               IF "MAX_VFDS" <> "MAX_ROOMS" * "MAX_RACKS_PER_ROOM" THEN
                   #bSettingsValid := FALSE;
                   #Status.ErrorMsg := CONCAT(IN1 := #Status.ErrorMsg, IN2 := ' MAX_VFDS != MAX_ROOMS*MAX_RACKS ');
               END_IF;

               IF #Controls.iSetNumRooms > "MAX_ROOMS" THEN
                   #bSettingsValid := FALSE;
                   #Status.ErrorMsg := CONCAT(IN1 := #Status.ErrorMsg, IN2 := ' NumRooms > MAX ');
               END_IF;

               FOR #i := 1 TO UINT_TO_INT("MAX_ROOMS") DO
                   IF #Controls.arrSetNumRacksPerRoom[#i] > "MAX_RACKS_PER_ROOM" THEN
                       #bSettingsValid := FALSE;
                       #Status.ErrorMsg := CONCAT(IN1 := #Status.ErrorMsg, IN2 := ' NumRacks > MAX ');
                       EXIT;
                   END_IF;
               END_FOR;

               IF "MAX_AI_PER_ROOM" <> ("NUM_AI_ROOM" + "NUM_AI_RACK" * "MAX_RACKS_PER_ROOM" + "EXTRA_AI_PER_ROOM") OR ( "MAX_AI_PER_ROOM" MOD 4 <> 0) THEN
                   #bSettingsValid := FALSE;
                   #Status.ErrorMsg := CONCAT(IN1 := #Status.ErrorMsg, IN2 := ' MAX_AI_PER_ROOM incorrect ');
               END_IF;

               IF "MAX_DQ_PER_ROOM" <> ("NUM_DQ_ROOM" + "NUM_DQ_RACK" * "MAX_RACKS_PER_ROOM" + "EXTRA_DQ_PER_ROOM") OR ( "MAX_DQ_PER_ROOM" MOD 8 <> 0) THEN
                   #bSettingsValid := FALSE;
                   #Status.ErrorMsg := CONCAT(IN1 := #Status.ErrorMsg, IN2 := ' MAX_DQ_PER_ROOM incorrect ');
               END_IF;

           END_REGION

           IF #bSettingsValid THEN
               // set number of rooms
               #iNumRooms := #Controls.iSetNumRooms;

               FOR #iRoomIndex := 1 TO #iNumRooms DO
                   // set number of racks in each room
                   "dbMain".Room[#iRoomIndex].Config.iNumRacks := #Controls.arrSetNumRacksPerRoom[#iRoomIndex];
               END_FOR;

               #iNextStep := #eStep_SetUp;

           ELSE
               #iNextStep := #eStep_Error;

           END_IF;

       END_IF;

   END_REGION

   REGION 1: Set up params

       IF #iStep = #eStep_SetUp THEN

           REGION Map VFD IO device system constants
               // Populate temp array of system constants for all possible VFDs
               #arrIoDeviceIds[1] := "RackPumpVFD_1~PROFINET_interface~IODevice";
               #arrIoDeviceIds[2] := "RackPumpVFD_2~PROFINET_interface~IODevice";
               #arrIoDeviceIds[3] := "RackPumpVFD_3~PROFINET_interface~IODevice";
               #arrIoDeviceIds[4] := "RackPumpVFD_4~PROFINET_interface~IODevice";
               #arrIoDeviceIds[5] := "RackPumpVFD_5~PROFINET_interface~IODevice";
               #arrIoDeviceIds[6] := "RackPumpVFD_6~PROFINET_interface~IODevice";
               (*
               #arrIoDeviceIds[7] := "RackPumpVFD_7~PROFINET_interface~IODevice";
               #arrIoDeviceIds[8] := "RackPumpVFD_8~PROFINET_interface~IODevice";
               #arrIoDeviceIds[9] := "RackPumpVFD_9~PROFINET_interface~IODevice";
               #arrIoDeviceIds[10] := "RackPumpVFD_10~PROFINET_interface~IODevice";
               #arrIoDeviceIds[11] := "RackPumpVFD_11~PROFINET_interface~IODevice";
               #arrIoDeviceIds[12] := "RackPumpVFD_12~PROFINET_interface~IODevice";


               #arrIoDeviceIds[13] := "RackPumpVFD_13~PROFINET_interface~IODevice";
               #arrIoDeviceIds[14] := "RackPumpVFD_14~PROFINET_interface~IODevice";
               #arrIoDeviceIds[15] := "RackPumpVFD_15~PROFINET_interface~IODevice";
               #arrIoDeviceIds[16] := "RackPumpVFD_16~PROFINET_interface~IODevice";
               #arrIoDeviceIds[17] := "RackPumpVFD_17~PROFINET_interface~IODevice";
               #arrIoDeviceIds[18] := "RackPumpVFD_18~PROFINET_interface~IODevice";
               #arrIoDeviceIds[19] := "RackPumpVFD_19~PROFINET_interface~IODevice";
               #arrIoDeviceIds[20] := "RackPumpVFD_20~PROFINET_interface~IODevice";
               #arrIoDeviceIds[21] := "RackPumpVFD_21~PROFINET_interface~IODevice";
               #arrIoDeviceIds[22] := "RackPumpVFD_22~PROFINET_interface~IODevice";
               #arrIoDeviceIds[23] := "RackPumpVFD_23~PROFINET_interface~IODevice";
               #arrIoDeviceIds[24] := "RackPumpVFD_24~PROFINET_interface~IODevice";
               #arrIoDeviceIds[25] := "RackPumpVFD_25~PROFINET_interface~IODevice";
               #arrIoDeviceIds[26] := "RackPumpVFD_26~PROFINET_interface~IODevice";
               #arrIoDeviceIds[27] := "RackPumpVFD_27~PROFINET_interface~IODevice";
               #arrIoDeviceIds[28] := "RackPumpVFD_28~PROFINET_interface~IODevice";
               #arrIoDeviceIds[29] := "RackPumpVFD_29~PROFINET_interface~IODevice";
               #arrIoDeviceIds[30] := "RackPumpVFD_30~PROFINET_interface~IODevice";
               *)

           END_REGION

           REGION Map VFD telegram hw submodule system constants
               // Populate temp array of system constants for all possible VFDs
               #arrTelegrams[1] := "RackPumpVFD_1~PROFINET_interface~Free_telegram";
               #arrTelegrams[2] := "RackPumpVFD_2~PROFINET_interface~Free_telegram";
               #arrTelegrams[3] := "RackPumpVFD_3~PROFINET_interface~Free_telegram";
               #arrTelegrams[4] := "RackPumpVFD_4~PROFINET_interface~Free_telegram";
               #arrTelegrams[5] := "RackPumpVFD_5~PROFINET_interface~Free_telegram";
               #arrTelegrams[6] := "RackPumpVFD_6~PROFINET_interface~Free_telegram";
               (*
               #arrTelegrams[7] := "RackPumpVFD_7~PROFINET_interface~Free_telegram";
               #arrTelegrams[8] := "RackPumpVFD_8~PROFINET_interface~Free_telegram";
               #arrTelegrams[9] := "RackPumpVFD_9~PROFINET_interface~Free_telegram";
               #arrTelegrams[10] := "RackPumpVFD_10~PROFINET_interface~Free_telegram";
               #arrTelegrams[11] := "RackPumpVFD_11~PROFINET_interface~Free_telegram";
               #arrTelegrams[12] := "RackPumpVFD_12~PROFINET_interface~Free_telegram";


               #arrTelegrams[13] := "RackPumpVFD_13~PROFINET_interface~Free_telegram";
               #arrTelegrams[14] := "RackPumpVFD_14~PROFINET_interface~Free_telegram";
               #arrTelegrams[15] := "RackPumpVFD_15~PROFINET_interface~Free_telegram";
               #arrTelegrams[16] := "RackPumpVFD_16~PROFINET_interface~Free_telegram";
               #arrTelegrams[17] := "RackPumpVFD_17~PROFINET_interface~Free_telegram";
               #arrTelegrams[18] := "RackPumpVFD_18~PROFINET_interface~Free_telegram";
               #arrTelegrams[19] := "RackPumpVFD_19~PROFINET_interface~Free_telegram";
               #arrTelegrams[20] := "RackPumpVFD_20~PROFINET_interface~Free_telegram";
               #arrTelegrams[21] := "RackPumpVFD_21~PROFINET_interface~Free_telegram";
               #arrTelegrams[22] := "RackPumpVFD_22~PROFINET_interface~Free_telegram";
               #arrTelegrams[23] := "RackPumpVFD_23~PROFINET_interface~Free_telegram";
               #arrTelegrams[24] := "RackPumpVFD_24~PROFINET_interface~Free_telegram";
               #arrTelegrams[25] := "RackPumpVFD_25~PROFINET_interface~Free_telegram";
               #arrTelegrams[26] := "RackPumpVFD_26~PROFINET_interface~Free_telegram";
               #arrTelegrams[27] := "RackPumpVFD_27~PROFINET_interface~Free_telegram";
               #arrTelegrams[28] := "RackPumpVFD_28~PROFINET_interface~Free_telegram";
               #arrTelegrams[29] := "RackPumpVFD_29~PROFINET_interface~Free_telegram";
               #arrTelegrams[30] := "RackPumpVFD_30~PROFINET_interface~Free_telegram";
               *)

           END_REGION

           REGION Assign VFDs to racks, set up IO reconfig array

               #iVfdCount := 0;

               FOR #iRoomIndex := 1 TO #iNumRooms DO

                   // Assign VFDs to configured rooms and racks, only using the ones we need
                   // Link up the Hw_SubModule system constant for each VFD's Profinet telegram

                   FOR #iRackIndex := 1 TO #Controls.arrSetNumRacksPerRoom[#iRoomIndex] DO
                       #iVfdCount += 1;

                       "dbMain".Room[#iRoomIndex].Rack[#iRackIndex].Fertigation.Pump.fbVFD.hwInTelegram :=
                       #arrTelegrams[#iVfdCount];

                   END_FOR;

               END_FOR;

               // populate data record array for reconfig io fb
               #arrVfdDeviceConfig[-2] := 16#0100; // Version of the data record (1.0)
               #arrVfdDeviceConfig[-1] := INT_TO_WORD(#iVfdCount); // Number of IO devices to be activated

               // populate input array with IO device IDs for all the VFDs we are using
               FOR #i := 0 TO #iVfdCount-1 DO
                   #arrVfdDeviceConfig[#i] := UINT_TO_WORD(#arrIoDeviceIds[#i+1]);
               END_FOR;

               // zero out rest of array (zero port interconnections used since everything is defined in topology)
               FOR #i := #iVfdCount TO UINT_TO_INT("MAX_VFDS") DO
                   #arrVfdDeviceConfig[#i] := 0;
               END_FOR;

           END_REGION

           REGION Assign Modbus TCP HVAC servers to rooms
               FOR #i := 1 TO #iNumRooms DO

                   // Port and connection ID
                   "dbMain".Room[#i].HVAC.Config.ID := INT_TO_UINT(80 + #i);

                   // IP address
                   "dbMain".Room[#i].HVAC.Config.ModbusServerAddr.ADDR[1] := 10;
                   "dbMain".Room[#i].HVAC.Config.ModbusServerAddr.ADDR[2] := 1;
                   "dbMain".Room[#i].HVAC.Config.ModbusServerAddr.ADDR[3] := 0;
                   "dbMain".Room[#i].HVAC.Config.ModbusServerAddr.ADDR[4] := INT_TO_BYTE(19 + #i);

               END_FOR;
           END_REGION

           IF #bInSimulation THEN
               #iNextStep := #eStep_Done;
           ELSE
               #iNextStep := #eStep_Deactivate;
           END_IF;

       END_IF;
   END_REGION

   REGION Call ReconfigIOSystem FB

       CASE #iStep OF
           #eStep_Deactivate:
               #ReconfigIOSystem.REQ := TRUE;
               #ReconfigIOSystem.MODE := 1;
               IF #ReconfigIOSystem.DONE THEN
                   #iNextStep := #eStep_WaitForDeactivate;
               END_IF;

           #eStep_WaitForDeactivate:
               #ReconfigIOSystem.REQ := FALSE;
               #iNextStep := #eStep_Reconfig;

           #eStep_Reconfig:
               #ReconfigIOSystem.REQ := TRUE;
               #ReconfigIOSystem.MODE := 2;
               IF #ReconfigIOSystem.DONE THEN
                   #iNextStep := #eStep_WaitForReconfig;
               END_IF;

           #eStep_WaitForReconfig:
               #ReconfigIOSystem.REQ := FALSE;
               #iNextStep := #eStep_Restart;

           #eStep_Restart:
               #ReconfigIOSystem.REQ := TRUE;
               #ReconfigIOSystem.MODE := 3;
               IF #ReconfigIOSystem.DONE THEN
                   #iNextStep := #eStep_Done;
               END_IF;

           ELSE
               #ReconfigIOSystem.REQ := FALSE;
               #ReconfigIOSystem.MODE := 0;

       END_CASE;

       #ReconfigIOSystem(REQ := #ReconfigIOSystem.REQ,
                         MODE := #ReconfigIOSystem.MODE,
                         LADDR := "Local~PROFINET_interface_1",
                         CTRLREC := #arrVfdDeviceConfig,
                         STATUS => #ReconfigIOSystem.STATUS,
                         BUSY => #ReconfigIOSystem.BUSY,
                         DONE => #ReconfigIOSystem.DONE,
                         ERROR => #ReconfigIOSystem.ERROR);

       // catch and log error
       IF #ReconfigIOSystem.ERROR THEN
           #Status.ErrorMsg := CONCAT(IN1 := #Status.ErrorMsg, IN2 := ' ReconfigIO Error Code: ');
           #retVal := HTA(IN := #ReconfigIOSystem.STATUS, N := 4, OUT => #strErrorCode);
           #Status.ErrorMsg := CONCAT(IN1 := #Status.ErrorMsg, IN2 := #strErrorCode);

           #Status.ErrorMsg := CONCAT(IN1 := #Status.ErrorMsg, IN2 := ' On device: ');
           #retVal := HTA(IN := #ReconfigIOSystem.ERR_INFO, N := 2, OUT => #strErrorCode);
           #Status.ErrorMsg := CONCAT(IN1 := #Status.ErrorMsg, IN2 := #strErrorCode);

           #iNextStep := #eStep_Error;
       END_IF;

   END_REGION

   REGION Set status outputs
       #Status.bDone := #iStep = #eStep_Done;
       #Status.bBusy := #iStep <> #eStep_Done AND #iStep <> #eStep_Error;
       #Status.bError := #iStep = #eStep_Error;

   END_REGION

   // set step for next scan
   #iStep := #iNextStep;
END_FUNCTION_BLOCK

ORGANIZATION_BLOCK "Main"   // OB1, LAD, ProgramCycle
TITLE = "Main Program Sweep (Cycle)"
{ S7_Optimized_Access := 'TRUE' }
VERSION : 0.1
   VAR_INPUT
      Initial_Call : Bool;   // Initial call of this OB
      Remanence : Bool;   // =True, if remanent data are available
   END_VAR
BEGIN

REGION Network 1
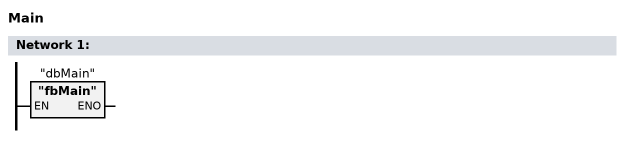
   RUNG wire#powerrail
      "dbMain"()
   END_RUNG
   // the same network as SCL:
   "dbMain"();   // "fbMain"
END_REGION
END_ORGANIZATION_BLOCK

// folder: Resources

FUNCTION_BLOCK "fbAlarmedSetpoint"   // FB1, LAD
{ S7_Optimized_Access := 'TRUE' }
VERSION : 0.1
// Processes raw analog input and evaluates alarms.
// Note: All alarms are momentary, i.e. no ack necessary and they reset themselves when the condition becomes false.
   VAR_INPUT
      iInRawValue : Int;
   END_VAR
   VAR RETAIN
      arrSetpoints : Array[1..10] of "udtTimeOfDaySetpoint";   // Setpoints need to be chronologically increasing
      rSetpoint : Real;
      rActual : Real;
      Alarms : Struct
         bHigh : Bool;   // rActual exceeds limit
         bLow : Bool;   // rActual exceeds limit
         bRate : Bool;   // rActual increases or decreases faster than the limit. False if rate is left as 0.
         bSetpoint : Bool;   // rActual does not reach rSetpoint within allowed time delay and deadband. False if deadband left at 0.
      END_STRUCT;
      Config : Struct
         rLowCalibration : Real := 0.0;
         rHighCalibration : Real := 100.0;
         Alarms : Struct
            rLowLimit : Real := 0.0;
            rHighLimit : Real := 100.0;
            rRateLimit : Real;   // Maximum permitted change in rActual per second
            rDeadband : Real;   // Range around rSetpoint that is still considered within range
            iSettlingSecs : Int;   // Allowable delay to allow rActual to reach rSetpoint after change
         END_STRUCT;
      END_STRUCT;
   END_VAR
   VAR
      TON_RateCheck : TON_TIME;
      rActual_Prev : Real;
      TON_Settling : TON_TIME;
      rSetpoint_Prev : Real;
   END_VAR
   VAR_TEMP
      localTime : Date_And_Time;
      ret_val : Int;
      currentTOD : Time_Of_Day;
      i : Int;
      currentTODsecs : DInt;
   END_VAR
BEGIN

REGION Network 1 (SCL): Scale raw input based on calibration
   #rActual := "fcAnalogInput"(iInRawValue := #iInRawValue,
                               rLowCalibration := #Config.rLowCalibration,
                               rHighCalibration := #Config.rHighCalibration);
END_REGION

REGION Network 2 (SCL): Low/high alarms
   #Alarms.bHigh := #rActual > #Config.Alarms.rHighLimit;
   #Alarms.bLow  := #rActual < #Config.Alarms.rLowLimit;
END_REGION

REGION Network 3 (SCL): Rate of change alarm
   // Set the current value on startup to prevent a spurious alarm
   IF "FirstScan" THEN
       #rActual_Prev := #rActual;
   END_IF;

   // Compare values at every given time interval to get rate of change
   IF #TON_RateCheck.Q THEN
       #Alarms.bRate := ( ABS(#rActual - #rActual_Prev) > #Config.Alarms.rRateLimit)
       AND (#Config.Alarms.rRateLimit <> 0.0); // ignore alarm if max rate is left at default of 0

       #rActual_Prev := #rActual;
   END_IF;

   #TON_RateCheck(IN := NOT #TON_RateCheck.Q,
                  PT := t#1s);
END_REGION

REGION Network 4: Get current time of day
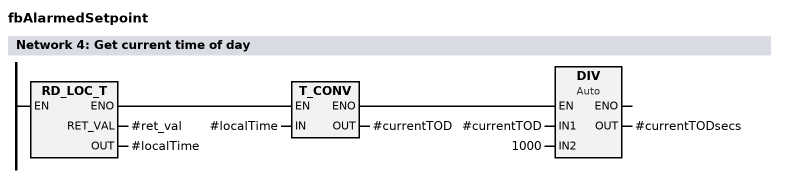
   // ENO of a box is taken as its EN; it also drops when the box reports an error
   #ret_val := RD_LOC_T(OUT => #localTime);
   #currentTOD := T_CONV(IN := #localTime);
   #currentTODsecs := #currentTOD / 1000;
END_REGION

REGION Network 5 (SCL): Determine current setpoint based on time of day
   IF #arrSetpoints[1].TimeOfDaySeconds = -1 THEN
       // If no time schedule is defined, default to first setpoint in array
       #rSetpoint := #arrSetpoints[1].rSetpoint;

   ELSIF #currentTODsecs < #arrSetpoints[1].TimeOfDaySeconds THEN
       // Check for setpoint from previous day
       FOR #i := 10 TO 1 BY -1 DO
           IF #arrSetpoints[#i].TimeOfDaySeconds <> -1 THEN
               #rSetpoint := #arrSetpoints[#i].rSetpoint;
               EXIT;
           END_IF;
       END_FOR;

   ELSE
       // Iterate through and find current setpoint
       FOR #i := 1 TO 9 DO
           IF #currentTODsecs < #arrSetpoints[#i + 1].TimeOfDaySeconds OR #arrSetpoints[#i + 1].TimeOfDaySeconds = -1 THEN
               #rSetpoint := #arrSetpoints[#i].rSetpoint;
               EXIT;
           ELSIF #i = 9 THEN
               #rSetpoint := #arrSetpoints[10].rSetpoint;
           END_IF;
       END_FOR;

   END_IF;
END_REGION

REGION Network 6 (SCL): Setpoint not reached alarm


   // Set the current value on startup to prevent a spurious alarm
   IF "FirstScan" THEN
       #rSetpoint_Prev := #rSetpoint;
   END_IF;

   // Evaluate alarm after settling time has elapsed
   #TON_Settling(IN := (#rSetpoint = #rSetpoint_Prev), // restart timer when setpoint changes
                 PT := INT_TO_TIME(#Config.Alarms.iSettlingSecs * 1000)); // convert to ms

   #Alarms.bSetpoint := #TON_Settling.Q AND (
   (#rActual < #rSetpoint - #Config.Alarms.rDeadband / 2.0) OR
   (#rActual > #rSetpoint + #Config.Alarms.rDeadband / 2.0) )
   AND (#Config.Alarms.rDeadband <> 0.0); // ignore alarm if deadband is left at default of 0

   // Save setpoint value for next comparison
   #rSetpoint_Prev := #rSetpoint;
END_REGION
END_FUNCTION_BLOCK

FUNCTION_BLOCK "fbModbusTCPClient"   // FB12, LAD
{ S7_Optimized_Access := 'TRUE' }
VERSION : 0.1
   VAR_INPUT
      bInRequest : Bool;
      bInReset : Bool;
      iInSlaveId : UInt;
   END_VAR
   VAR_OUTPUT
      bOutError : Bool;
      wOutLastErrorCode : Word;
   END_VAR
   VAR_IN_OUT
      InOutConnect : TCON_IP_v4;
      InOutReadDiscreteData : Array[*] of "udtModbusValBool";
      InOutWriteCoilData : Array[*] of "udtModbusValBool";
      InOutReadRegisterData : Array[*] of "udtModbusValReal";
      InOutWriteRegisterData : Array[*] of "udtModbusValReal";
   END_VAR
   VAR
      iState : Int;
      iNextState : Int;
      insModbusClient_TCP : MB_CLIENT;
      bTrigReset : Bool;
      bTrigReq : Bool;
      iNumReadRegisters : DInt;
      iNumWriteRegisters : DInt;
      iCurrentRegisterReadIndex : DInt;
      iCurrentRegisterWriteIndex : DInt;
      arrDataWords : Array[0..1] of Word;
      iNumReadDiscrete : DInt;
      iCurrentDiscreteReadIndex : DInt;
      iCurrentCoilWriteIndex : DInt;
      iNumWriteCoils : DInt;
   END_VAR
   VAR_TEMP
      iMode : USInt;
      iDataAddr : UDInt;
      tempDWord : DWord;
      bConnect : Bool;
      rTemp : Real;
   END_VAR
   VAR CONSTANT
      MODE_READ : USInt := 0;
      MODE_WRITE : USInt := 1;
      IDLE : Int := 0;
      READ_DISC_INIT : Int := 100;
      READ_DISC : Int := 110;
      READ_DISC_NEXT : Int := 120;
      WRITE_COILS_INIT : Int := 200;
      WRITE_COILS : Int := 210;
      WRITE_COILS_NEXT : Int := 220;
      READ_REGS_INIT : Int := 300;
      READ_REGS : Int := 310;
      READ_REGS_PARSE : Int := 320;
      READ_REGS_NEXT : Int := 330;
      WRITE_REGS_INIT : Int := 400;
      WRITE_REGS : Int := 410;
      WRITE_REGS_READBACK_INIT : Int := 420;
      WRITE_REGS_READBACK : Int := 430;
      WRITE_REGS_READBACK_PARSE : Int := 440;
      WRITE_REGS_NEXT : Int := 450;
   END_VAR
   VAR_TEMP   // added for the SCL form of the ladder/FBD networks
      _w1 : Bool;
      _w2 : Bool;
      _w3 : Bool;
      _w4 : Bool;
      _w5 : Bool;
      _w6 : Bool;
      _w7 : Bool;
      _w8 : Bool;
   END_VAR
BEGIN

REGION Network 1: ------------------------------ State Logic ----------------------------------
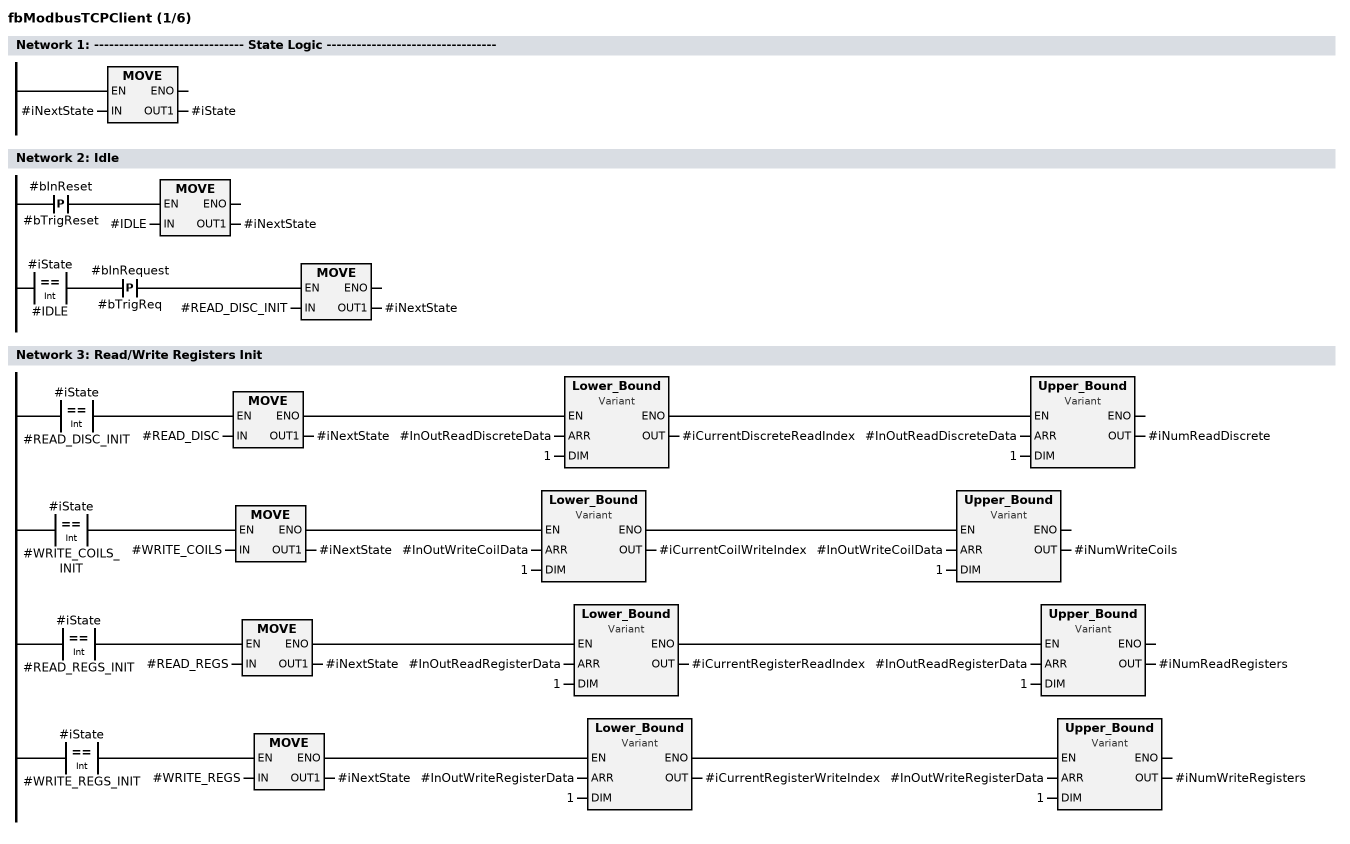
   RUNG wire#powerrail
      Move(in := #iNextState, out1 => #iState)
   END_RUNG
   // the same network as SCL:
   #iState := #iNextState;
END_REGION

REGION Network 2: Idle
   RUNG wire#powerrail
      P_Contact(operand := #bInReset, bit := #bTrigReset)
      Move(in := #IDLE, out1 => #iNextState)
   END_RUNG
   RUNG wire#powerrail
      { S7_Templates := "SrcType := Int" } EQ_Contact(in1 := #iState, in2 := #IDLE)
      P_Contact(operand := #bInRequest, bit := #bTrigReq)
      Move(in := #READ_DISC_INIT, out1 => #iNextState)
   END_RUNG
   // the same network as SCL:
   #_w1 := #bInReset AND NOT #bTrigReset;   // rising edge of #bInReset
   #bTrigReset := #bInReset;
   IF #_w1 THEN #iNextState := #IDLE; END_IF;
   #_w2 := (#iState = #IDLE) AND #bInRequest AND NOT #bTrigReq;   // rising edge of #bInRequest
   #bTrigReq := #bInRequest;
   IF #_w2 THEN #iNextState := #READ_DISC_INIT; END_IF;
END_REGION

REGION Network 3: Read/Write Registers Init
   // no SCL statement known for Lower_Bound, Upper_Bound: written as a call
   // ENO of a box is taken as its EN; it also drops when the box reports an error
   IF #iState = #READ_DISC_INIT THEN
       #iNextState := #READ_DISC;
       Lower_Bound(arr := #InOutReadDiscreteData, dim := 1, out => #iCurrentDiscreteReadIndex);
       Upper_Bound(arr := #InOutReadDiscreteData, dim := 1, out => #iNumReadDiscrete);
   END_IF;
   IF #iState = #WRITE_COILS_INIT THEN
       #iNextState := #WRITE_COILS;
       Lower_Bound(arr := #InOutWriteCoilData, dim := 1, out => #iCurrentCoilWriteIndex);
       Upper_Bound(arr := #InOutWriteCoilData, dim := 1, out => #iNumWriteCoils);
   END_IF;
   IF #iState = #READ_REGS_INIT THEN
       #iNextState := #READ_REGS;
       Lower_Bound(arr := #InOutReadRegisterData, dim := 1, out => #iCurrentRegisterReadIndex);
       Upper_Bound(arr := #InOutReadRegisterData, dim := 1, out => #iNumReadRegisters);
   END_IF;
   IF #iState = #WRITE_REGS_INIT THEN
       #iNextState := #WRITE_REGS;
       Lower_Bound(arr := #InOutWriteRegisterData, dim := 1, out => #iCurrentRegisterWriteIndex);
       Upper_Bound(arr := #InOutWriteRegisterData, dim := 1, out => #iNumWriteRegisters);
   END_IF;
END_REGION

REGION Network 4: Wait for Read/Write to be done
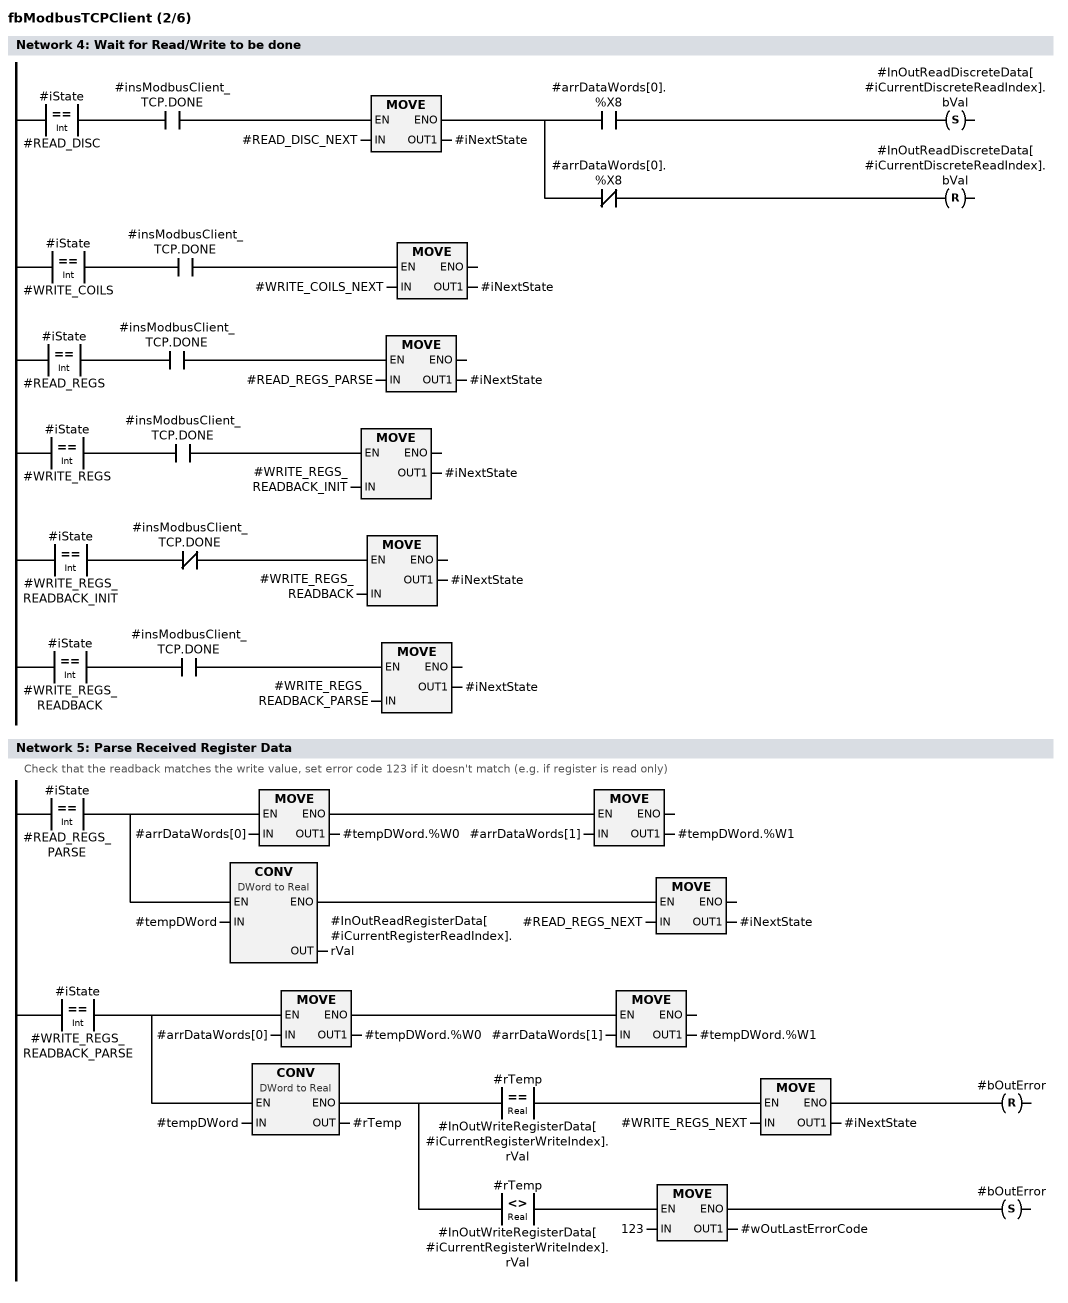
   RUNG wire#powerrail
      { S7_Templates := "SrcType := Int" } EQ_Contact(in1 := #iState, in2 := #READ_DISC)
      Contact( #insModbusClient_TCP.DONE )
      Move(in := #READ_DISC_NEXT, out1 => #iNextState)
      wire#w1
      Contact( #arrDataWords[0].%X8 )
      S_Coil( #InOutReadDiscreteData[#iCurrentDiscreteReadIndex].bVal )
   END_RUNG
   RUNG wire#w1
      I_Contact( #arrDataWords[0].%X8 )
      R_Coil( #InOutReadDiscreteData[#iCurrentDiscreteReadIndex].bVal )
   END_RUNG
   RUNG wire#powerrail
      { S7_Templates := "SrcType := Int" } EQ_Contact(in1 := #iState, in2 := #WRITE_COILS)
      Contact( #insModbusClient_TCP.DONE )
      Move(in := #WRITE_COILS_NEXT, out1 => #iNextState)
   END_RUNG
   RUNG wire#powerrail
      { S7_Templates := "SrcType := Int" } EQ_Contact(in1 := #iState, in2 := #READ_REGS)
      Contact( #insModbusClient_TCP.DONE )
      Move(in := #READ_REGS_PARSE, out1 => #iNextState)
   END_RUNG
   RUNG wire#powerrail
      { S7_Templates := "SrcType := Int" } EQ_Contact(in1 := #iState, in2 := #WRITE_REGS)
      Contact( #insModbusClient_TCP.DONE )
      Move(in := #WRITE_REGS_READBACK_INIT, out1 => #iNextState)
   END_RUNG
   RUNG wire#powerrail
      { S7_Templates := "SrcType := Int" } EQ_Contact(in1 := #iState, in2 := #WRITE_REGS_READBACK_INIT)
      I_Contact( #insModbusClient_TCP.DONE )
      Move(in := #WRITE_REGS_READBACK, out1 => #iNextState)
   END_RUNG
   RUNG wire#powerrail
      { S7_Templates := "SrcType := Int" } EQ_Contact(in1 := #iState, in2 := #WRITE_REGS_READBACK)
      Contact( #insModbusClient_TCP.DONE )
      Move(in := #WRITE_REGS_READBACK_PARSE, out1 => #iNextState)
   END_RUNG
   // the same network as SCL:
   #_w1 := (#iState = #READ_DISC) AND #insModbusClient_TCP.DONE;
   IF #_w1 THEN #iNextState := #READ_DISC_NEXT; END_IF;
   IF #_w1 AND #arrDataWords[0].%X8 THEN
       #InOutReadDiscreteData[#iCurrentDiscreteReadIndex].bVal := TRUE;
   END_IF;
   IF #_w1 AND NOT #arrDataWords[0].%X8 THEN
       #InOutReadDiscreteData[#iCurrentDiscreteReadIndex].bVal := FALSE;
   END_IF;
   IF (#iState = #WRITE_COILS) AND #insModbusClient_TCP.DONE THEN #iNextState := #WRITE_COILS_NEXT; END_IF;
   IF (#iState = #READ_REGS) AND #insModbusClient_TCP.DONE THEN #iNextState := #READ_REGS_PARSE; END_IF;
   IF (#iState = #WRITE_REGS) AND #insModbusClient_TCP.DONE THEN
       #iNextState := #WRITE_REGS_READBACK_INIT;
   END_IF;
   IF (#iState = #WRITE_REGS_READBACK_INIT) AND NOT #insModbusClient_TCP.DONE THEN
       #iNextState := #WRITE_REGS_READBACK;
   END_IF;
   IF (#iState = #WRITE_REGS_READBACK) AND #insModbusClient_TCP.DONE THEN
       #iNextState := #WRITE_REGS_READBACK_PARSE;
   END_IF;
END_REGION

REGION Network 5: Parse Received Register Data
   // Check that the readback matches the write value, set error code 123 if it doesn't match (e.g. if register is read only)
   RUNG wire#powerrail
      { S7_Templates := "SrcType := Int" } EQ_Contact(in1 := #iState, in2 := #READ_REGS_PARSE)
      wire#w1
      Move(in := #arrDataWords[0], out1 => #tempDWord.%W0)
      Move(in := #arrDataWords[1], out1 => #tempDWord.%W1)
   END_RUNG
   RUNG wire#w1
      { S7_Templates := "[SrcType := DWord, DestType := Real]" } Convert(in := #tempDWord, out => #InOutReadRegisterData[#iCurrentRegisterReadIndex].rVal)
      Move(in := #READ_REGS_NEXT, out1 => #iNextState)
   END_RUNG
   RUNG wire#powerrail
      { S7_Templates := "SrcType := Int" } EQ_Contact(in1 := #iState, in2 := #WRITE_REGS_READBACK_PARSE)
      wire#w2
      Move(in := #arrDataWords[0], out1 => #tempDWord.%W0)
      Move(in := #arrDataWords[1], out1 => #tempDWord.%W1)
   END_RUNG
   RUNG wire#w2
      { S7_Templates := "[SrcType := DWord, DestType := Real]" } Convert(in := #tempDWord, out => #rTemp)
      wire#w3
      { S7_Templates := "SrcType := Real" } EQ_Contact(in1 := #rTemp, in2 := #InOutWriteRegisterData[#iCurrentRegisterWriteIndex].rVal)
      Move(in := #WRITE_REGS_NEXT, out1 => #iNextState)
      R_Coil( #bOutError )
   END_RUNG
   RUNG wire#w3
      { S7_Templates := "SrcType := Real" } NE_Contact(in1 := #rTemp, in2 := #InOutWriteRegisterData[#iCurrentRegisterWriteIndex].rVal)
      Move(in := 123, out1 => #wOutLastErrorCode)
      S_Coil( #bOutError )
   END_RUNG
   // the same network as SCL:
   IF #iState = #READ_REGS_PARSE THEN
       #tempDWord.%W0 := #arrDataWords[0];
       #tempDWord.%W1 := #arrDataWords[1];
       #InOutReadRegisterData[#iCurrentRegisterReadIndex].rVal := DWORD_TO_REAL(#tempDWord);
       #iNextState := #READ_REGS_NEXT;
   END_IF;
   #_w1 := #iState = #WRITE_REGS_READBACK_PARSE;
   IF #_w1 THEN
       #tempDWord.%W0 := #arrDataWords[0];
       #tempDWord.%W1 := #arrDataWords[1];
       #rTemp := DWORD_TO_REAL(#tempDWord);
   END_IF;
   IF #_w1 AND (#rTemp = #InOutWriteRegisterData[#iCurrentRegisterWriteIndex].rVal) THEN
       #iNextState := #WRITE_REGS_NEXT;
       #bOutError := FALSE;
   END_IF;
   IF #_w1 AND (#rTemp <> #InOutWriteRegisterData[#iCurrentRegisterWriteIndex].rVal) THEN
       #wOutLastErrorCode := 123;
       #bOutError := TRUE;
   END_IF;
END_REGION

REGION Network 6: Move on to next address
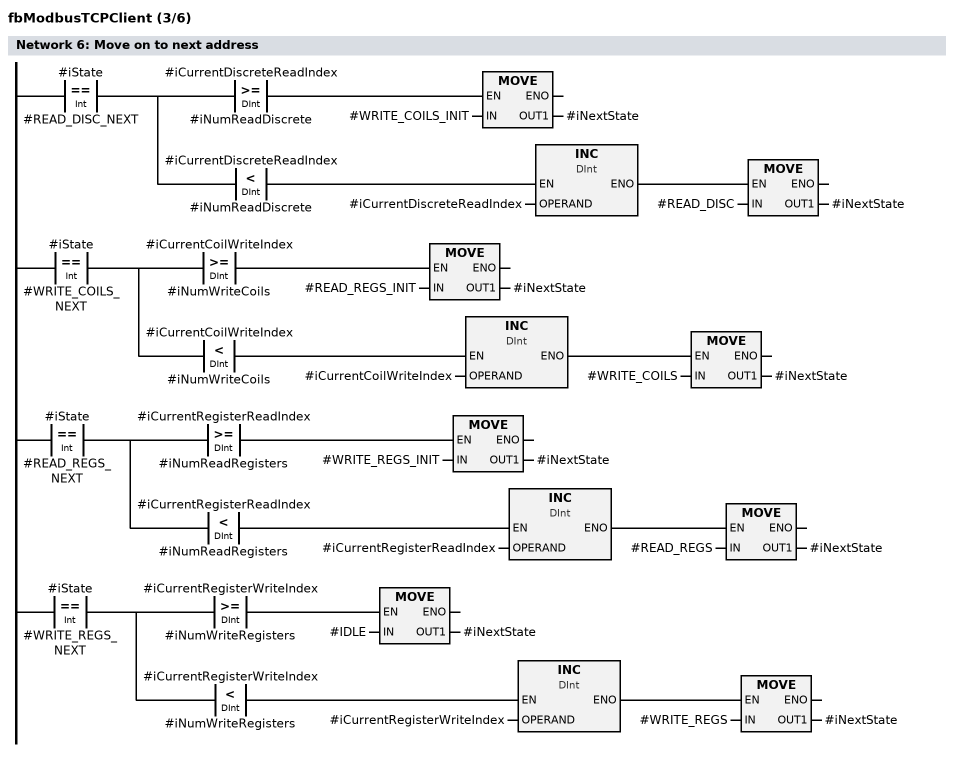
   RUNG wire#powerrail
      { S7_Templates := "SrcType := Int" } EQ_Contact(in1 := #iState, in2 := #READ_DISC_NEXT)
      wire#w1
      { S7_Templates := "SrcType := DInt" } GE_Contact(in1 := #iCurrentDiscreteReadIndex, in2 := #iNumReadDiscrete)
      Move(in := #WRITE_COILS_INIT, out1 => #iNextState)
   END_RUNG
   RUNG wire#w1
      { S7_Templates := "SrcType := DInt" } LT_Contact(in1 := #iCurrentDiscreteReadIndex, in2 := #iNumReadDiscrete)
      { S7_Templates := "DestType := DInt" } Inc( #iCurrentDiscreteReadIndex )
      Move(in := #READ_DISC, out1 => #iNextState)
   END_RUNG
   RUNG wire#powerrail
      { S7_Templates := "SrcType := Int" } EQ_Contact(in1 := #iState, in2 := #WRITE_COILS_NEXT)
      wire#w2
      { S7_Templates := "SrcType := DInt" } GE_Contact(in1 := #iCurrentCoilWriteIndex, in2 := #iNumWriteCoils)
      Move(in := #READ_REGS_INIT, out1 => #iNextState)
   END_RUNG
   RUNG wire#w2
      { S7_Templates := "SrcType := DInt" } LT_Contact(in1 := #iCurrentCoilWriteIndex, in2 := #iNumWriteCoils)
      { S7_Templates := "DestType := DInt" } Inc( #iCurrentCoilWriteIndex )
      Move(in := #WRITE_COILS, out1 => #iNextState)
   END_RUNG
   RUNG wire#powerrail
      { S7_Templates := "SrcType := Int" } EQ_Contact(in1 := #iState, in2 := #READ_REGS_NEXT)
      wire#w3
      { S7_Templates := "SrcType := DInt" } GE_Contact(in1 := #iCurrentRegisterReadIndex, in2 := #iNumReadRegisters)
      Move(in := #WRITE_REGS_INIT, out1 => #iNextState)
   END_RUNG
   RUNG wire#w3
      { S7_Templates := "SrcType := DInt" } LT_Contact(in1 := #iCurrentRegisterReadIndex, in2 := #iNumReadRegisters)
      { S7_Templates := "DestType := DInt" } Inc( #iCurrentRegisterReadIndex )
      Move(in := #READ_REGS, out1 => #iNextState)
   END_RUNG
   RUNG wire#powerrail
      { S7_Templates := "SrcType := Int" } EQ_Contact(in1 := #iState, in2 := #WRITE_REGS_NEXT)
      wire#w4
      { S7_Templates := "SrcType := DInt" } GE_Contact(in1 := #iCurrentRegisterWriteIndex, in2 := #iNumWriteRegisters)
      Move(in := #IDLE, out1 => #iNextState)
   END_RUNG
   RUNG wire#w4
      { S7_Templates := "SrcType := DInt" } LT_Contact(in1 := #iCurrentRegisterWriteIndex, in2 := #iNumWriteRegisters)
      { S7_Templates := "DestType := DInt" } Inc( #iCurrentRegisterWriteIndex )
      Move(in := #WRITE_REGS, out1 => #iNextState)
   END_RUNG
   // the same network as SCL:
   #_w1 := #iState = #READ_DISC_NEXT;
   IF #_w1 AND (#iCurrentDiscreteReadIndex >= #iNumReadDiscrete) THEN
       #iNextState := #WRITE_COILS_INIT;
   END_IF;
   #_w2 := #_w1 AND (#iCurrentDiscreteReadIndex < #iNumReadDiscrete);
   IF #_w2 THEN
       #iCurrentDiscreteReadIndex := #iCurrentDiscreteReadIndex + 1;
       #iNextState := #READ_DISC;
   END_IF;
   #_w3 := #iState = #WRITE_COILS_NEXT;
   IF #_w3 AND (#iCurrentCoilWriteIndex >= #iNumWriteCoils) THEN #iNextState := #READ_REGS_INIT; END_IF;
   #_w4 := #_w3 AND (#iCurrentCoilWriteIndex < #iNumWriteCoils);
   IF #_w4 THEN
       #iCurrentCoilWriteIndex := #iCurrentCoilWriteIndex + 1;
       #iNextState := #WRITE_COILS;
   END_IF;
   #_w5 := #iState = #READ_REGS_NEXT;
   IF #_w5 AND (#iCurrentRegisterReadIndex >= #iNumReadRegisters) THEN
       #iNextState := #WRITE_REGS_INIT;
   END_IF;
   #_w6 := #_w5 AND (#iCurrentRegisterReadIndex < #iNumReadRegisters);
   IF #_w6 THEN
       #iCurrentRegisterReadIndex := #iCurrentRegisterReadIndex + 1;
       #iNextState := #READ_REGS;
   END_IF;
   #_w7 := #iState = #WRITE_REGS_NEXT;
   IF #_w7 AND (#iCurrentRegisterWriteIndex >= #iNumWriteRegisters) THEN #iNextState := #IDLE; END_IF;
   #_w8 := #_w7 AND (#iCurrentRegisterWriteIndex < #iNumWriteRegisters);
   IF #_w8 THEN
       #iCurrentRegisterWriteIndex := #iCurrentRegisterWriteIndex + 1;
       #iNextState := #WRITE_REGS;
   END_IF;
END_REGION

REGION Network 7: ------------------------------ Configure settings and call MB_CLIENT ----------------------------------
END_REGION

REGION Network 8: Set register and data bytes based on array index
   // Assuming that all input address data is formatted with full Modbus address offsets, i.e. coils (00001), discrete inputs (10001), input registers (30001), holding registers (40001)
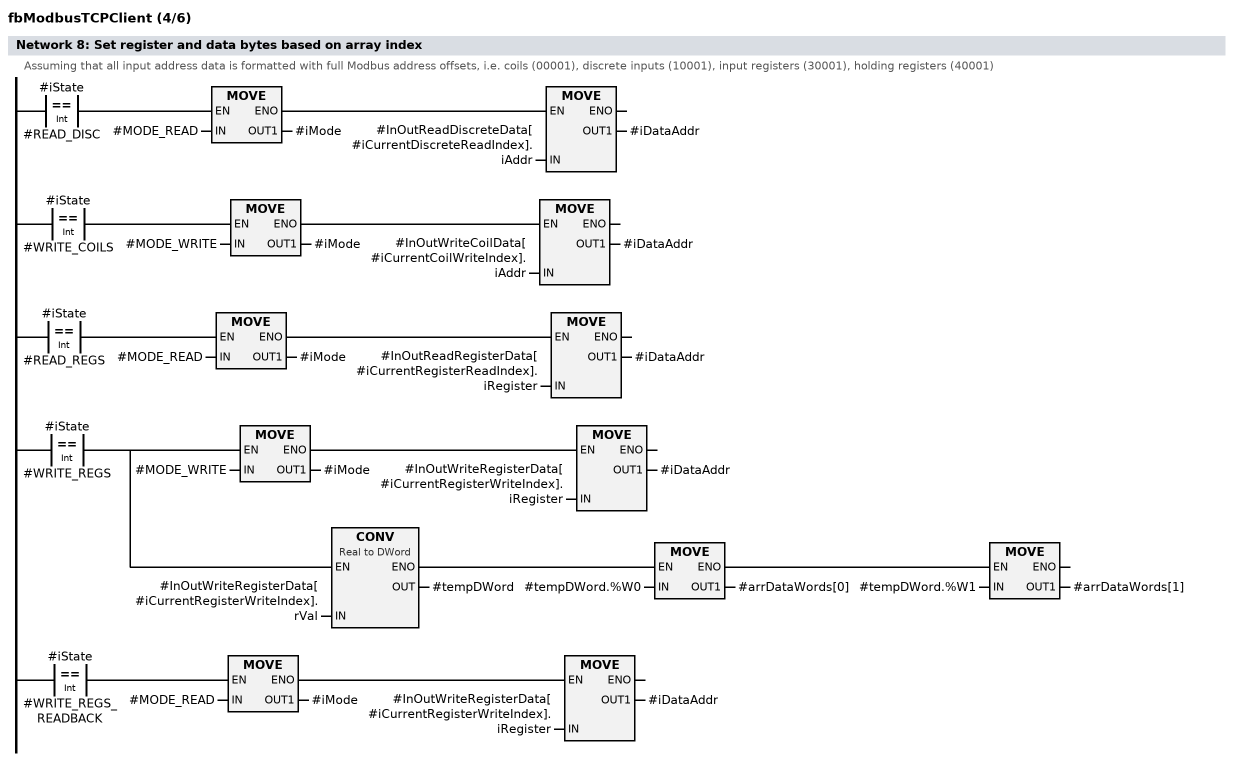
   RUNG wire#powerrail
      { S7_Templates := "SrcType := Int" } EQ_Contact(in1 := #iState, in2 := #READ_DISC)
      Move(in := #MODE_READ, out1 => #iMode)
      Move(in := #InOutReadDiscreteData[#iCurrentDiscreteReadIndex].iAddr, out1 => #iDataAddr)
   END_RUNG
   RUNG wire#powerrail
      { S7_Templates := "SrcType := Int" } EQ_Contact(in1 := #iState, in2 := #WRITE_COILS)
      Move(in := #MODE_WRITE, out1 => #iMode)
      Move(in := #InOutWriteCoilData[#iCurrentCoilWriteIndex].iAddr, out1 => #iDataAddr)
   END_RUNG
   RUNG wire#powerrail
      { S7_Templates := "SrcType := Int" } EQ_Contact(in1 := #iState, in2 := #READ_REGS)
      Move(in := #MODE_READ, out1 => #iMode)
      Move(in := #InOutReadRegisterData[#iCurrentRegisterReadIndex].iRegister, out1 => #iDataAddr)
   END_RUNG
   RUNG wire#powerrail
      { S7_Templates := "SrcType := Int" } EQ_Contact(in1 := #iState, in2 := #WRITE_REGS)
      wire#w1
      Move(in := #MODE_WRITE, out1 => #iMode)
      Move(in := #InOutWriteRegisterData[#iCurrentRegisterWriteIndex].iRegister, out1 => #iDataAddr)
   END_RUNG
   RUNG wire#w1
      { S7_Templates := "[SrcType := Real, DestType := DWord]" } Convert(in := #InOutWriteRegisterData[#iCurrentRegisterWriteIndex].rVal, out => #tempDWord)
      Move(in := #tempDWord.%W0, out1 => #arrDataWords[0])
      Move(in := #tempDWord.%W1, out1 => #arrDataWords[1])
   END_RUNG
   RUNG wire#powerrail
      { S7_Templates := "SrcType := Int" } EQ_Contact(in1 := #iState, in2 := #WRITE_REGS_READBACK)
      Move(in := #MODE_READ, out1 => #iMode)
      Move(in := #InOutWriteRegisterData[#iCurrentRegisterWriteIndex].iRegister, out1 => #iDataAddr)
   END_RUNG
   // the same network as SCL:
   IF #iState = #READ_DISC THEN
       #iMode := #MODE_READ;
       #iDataAddr := #InOutReadDiscreteData[#iCurrentDiscreteReadIndex].iAddr;
   END_IF;
   IF #iState = #WRITE_COILS THEN
       #iMode := #MODE_WRITE;
       #iDataAddr := #InOutWriteCoilData[#iCurrentCoilWriteIndex].iAddr;
   END_IF;
   IF #iState = #READ_REGS THEN
       #iMode := #MODE_READ;
       #iDataAddr := #InOutReadRegisterData[#iCurrentRegisterReadIndex].iRegister;
   END_IF;
   IF #iState = #WRITE_REGS THEN
       #iMode := #MODE_WRITE;
       #iDataAddr := #InOutWriteRegisterData[#iCurrentRegisterWriteIndex].iRegister;
       #tempDWord := REAL_TO_DWORD(#InOutWriteRegisterData[#iCurrentRegisterWriteIndex].rVal);
       #arrDataWords[0] := #tempDWord.%W0;
       #arrDataWords[1] := #tempDWord.%W1;
   END_IF;
   IF #iState = #WRITE_REGS_READBACK THEN
       #iMode := #MODE_READ;
       #iDataAddr := #InOutWriteRegisterData[#iCurrentRegisterWriteIndex].iRegister;
   END_IF;
END_REGION

REGION Network 9: MB_CLIENT block call
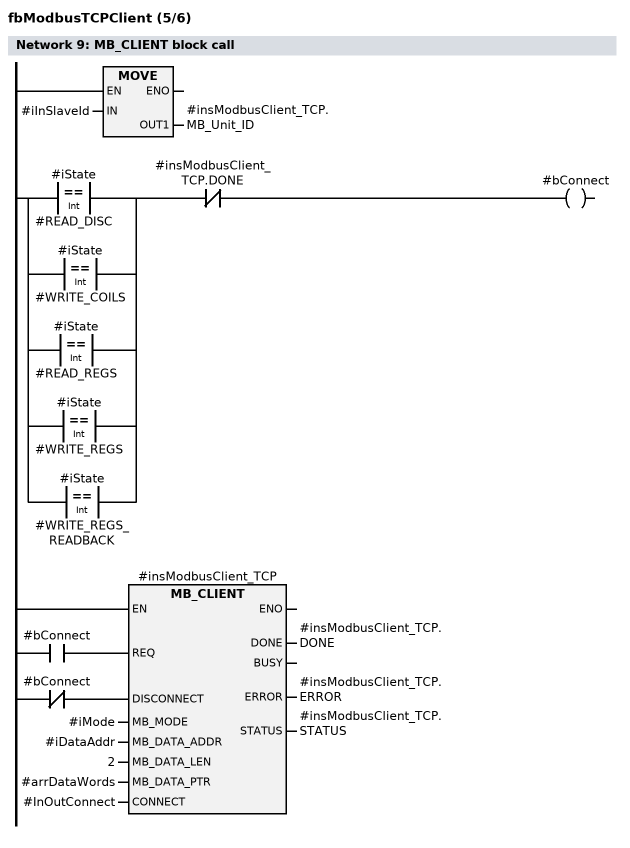
   #insModbusClient_TCP.MB_Unit_ID := #iInSlaveId;
   #bConnect := ((#iState = #READ_DISC) OR (#iState = #WRITE_COILS) OR (#iState = #READ_REGS) OR (#iState = #WRITE_REGS) OR (#iState = #WRITE_REGS_READBACK)) AND NOT #insModbusClient_TCP.DONE;
   #insModbusClient_TCP(REQ := #bConnect,   // MB_CLIENT
                        DISCONNECT := NOT #bConnect,
                        MB_MODE := #iMode,
                        MB_DATA_ADDR := #iDataAddr,
                        MB_DATA_LEN := 2,
                        MB_DATA_PTR := #arrDataWords,
                        CONNECT := #InOutConnect,
                        DONE => #insModbusClient_TCP.DONE,
                        ERROR => #insModbusClient_TCP.ERROR,
                        STATUS => #insModbusClient_TCP.STATUS);
END_REGION

REGION Network 10: Set error status
   // Ignore error code 16#80A3 (same connection already being used)
   // Go back to idle if stuck waiting for read/write
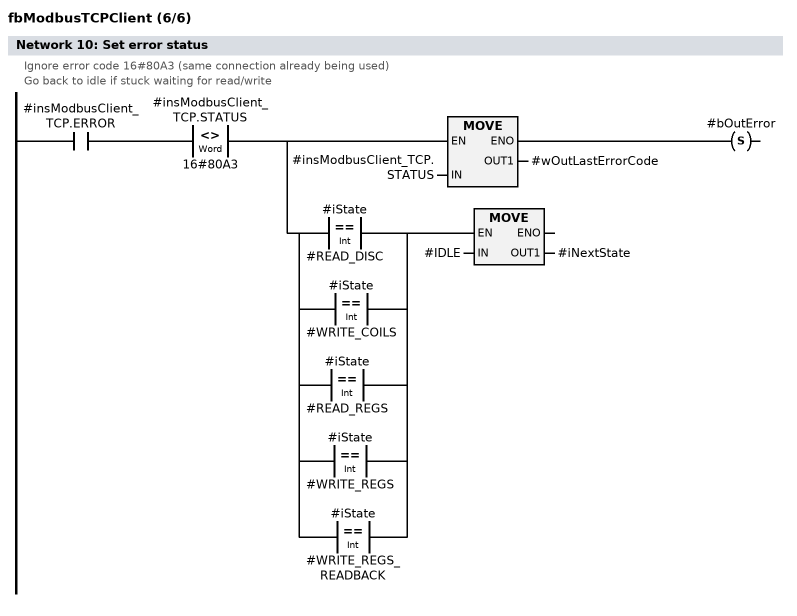
   RUNG wire#powerrail
      Contact( #insModbusClient_TCP.ERROR )
      { S7_Templates := "SrcType := Word" } NE_Contact(in1 := #insModbusClient_TCP.STATUS, in2 := 16#80A3)
      wire#w1
      Move(in := #insModbusClient_TCP.STATUS, out1 => #wOutLastErrorCode)
      S_Coil( #bOutError )
   END_RUNG
   RUNG wire#w1
      { S7_Templates := "SrcType := Int" } EQ_Contact(in1 := #iState, in2 := #READ_DISC)
      wire#w2
      Move(in := #IDLE, out1 => #iNextState)
   END_RUNG
   RUNG wire#w1
      { S7_Templates := "SrcType := Int" } EQ_Contact(in1 := #iState, in2 := #WRITE_COILS)
   END_RUNG wire#w2
   RUNG wire#w1
      { S7_Templates := "SrcType := Int" } EQ_Contact(in1 := #iState, in2 := #READ_REGS)
   END_RUNG wire#w2
   RUNG wire#w1
      { S7_Templates := "SrcType := Int" } EQ_Contact(in1 := #iState, in2 := #WRITE_REGS)
   END_RUNG wire#w2
   RUNG wire#w1
      { S7_Templates := "SrcType := Int" } EQ_Contact(in1 := #iState, in2 := #WRITE_REGS_READBACK)
   END_RUNG wire#w2
   // the same network as SCL:
   #_w1 := #insModbusClient_TCP.ERROR AND (#insModbusClient_TCP.STATUS <> 16#80A3);
   IF #_w1 THEN
       #wOutLastErrorCode := #insModbusClient_TCP.STATUS;
       #bOutError := TRUE;
   END_IF;
   IF #_w1 AND ((#iState = #READ_DISC) OR (#iState = #WRITE_COILS) OR (#iState = #READ_REGS) OR (#iState = #WRITE_REGS) OR (#iState = #WRITE_REGS_READBACK)) THEN
       #iNextState := #IDLE;
   END_IF;
END_REGION
END_FUNCTION_BLOCK

FUNCTION "fcAnalogInput" : Real   // FC2, SCL
{ S7_Optimized_Access := 'TRUE' }
VERSION : 0.1
   VAR_INPUT
      iInRawValue : Int;
      rLowCalibration : Real;
      rHighCalibration : Real;
   END_VAR
BEGIN
   // Scale raw input (0 to 27648 for 4-20mA and 0-10V)
   #fcAnalogInput :=

   ( INT_TO_REAL(#iInRawValue) / INT_TO_REAL("IoScaling.S7Analog.Default.iRawMax")) *
   (#rHighCalibration - #rLowCalibration) + #rLowCalibration;
END_FUNCTION

FUNCTION "fcDigitalOutput" : Bool   // FC3, SCL
{ S7_Optimized_Access := 'TRUE' }
VERSION : 0.1
   VAR_INPUT
      bInAutoVal : Bool;   // Value automatically set by the program
   END_VAR
   VAR_IN_OUT
      InOutUdt : "udtDigitalOutput";
   END_VAR
   // Ret_Val : Retrurn value to write to physical output
BEGIN

   IF #InOutUdt.bOverrideEnable THEN
       // if override is active, use override vallue
       #InOutUdt.bStatus := #InOutUdt.bOverrideVal;
   ELSE
       // if override is not active, make override value track auto
       // so that simply activating override mode does not
       // change the output value
       #InOutUdt.bOverrideVal := #bInAutoVal;
       #InOutUdt.bStatus := #bInAutoVal;
   END_IF;

   // map requested auto value to udt for monitoring
   #InOutUdt.bAutoVal := #bInAutoVal;

   // set FC return value for actual physical output
   #fcDigitalOutput := #InOutUdt.bStatus;
END_FUNCTION

// folder: Resources/fbVFD

FUNCTION_BLOCK "fbVFD_GSeries"   // FB120, LAD
TITLE = Controls a Siemens G120 VFD (or MicroMaster)
{ S7_Optimized_Access := 'TRUE' }
VERSION : 0.1
   VAR_INPUT
      tInTimeout : Time;   // Timeout Time
      iInMode : Int;   // Mode Selection
      hwInTelegram : Hw_SubModule;   // VFD Standard Telegram 1 HW address
      bInEstop : Bool;   // Estop
      bInSignalContactor : Bool;   // Feedback signal from Contactor
      bInEnableForward : Bool;   // Forward motion enebled
      bInEnableReverse : Bool := false;   // Reverse motion enabled
      rInCommandSpeed : Real;   // Auto mode speed SP
      bInCommandForward : Bool;   // Move forward in automatic mode
      bInCommandReverse : Bool := false;   // Move Reverse in automatic mode
      bInResetError : Bool;   // Reset Error
      bInMotorProtector : Bool := true;   // Motor Protector input
      bInLocalDisconnect : Bool := true;   // Local switch input
      bInClutch : Bool := true;   // Overload clutch
      bInCoolingFan : Bool := true;   // Cooling fan input
      bInUseCurrentAlarm : Bool := false;   // True if current alarm should be active
      bInUseMaxFrequencyAlarm : Bool := false;   // True is max frequency alarm should be active
      bInSimulate : Bool := false;   // Activate device simulation
   END_VAR
   VAR_OUTPUT
      rOutSpeed : Real;   // Actual motor speed
      bOutContactor : Bool;   // Motor contactor ON
      bOutCommandForward : Bool;   // Motor forward command
      bOutCommandReverse : Bool := false;   // Motor reverse command
      bOutActiveForward : Bool;   // Motor is running forward
      bOutActiveReverse : Bool;   // Motor is running backward
      bOutAuto : Bool;   // Block in auto mode
      bOutError : Bool;   // Error exists
      ERROR_VFD : "udtError_VFD";   // UDT Structure for VFD errors
   END_VAR
   VAR_IN_OUT
      HMI_VFD_Control : "udtHMI_VFD_Control";   // UDT Structure for VFD HMI control
   END_VAR
   VAR
      ErrorScroller : "fbErrorScroller";   // fb to control scrolling of errors on HMI
      TON_TimeOut : TON_TIME;   // Timer for Timeout time
      TON_ContactorDelay : TON_TIME;   // Contactor on delay timer before check errors
      TON_CoolingFan : TON_TIME;
      TON_CurrentLimitDebounce : TON_TIME;   // Debounce timer for current at limit
      iLastMode : Int;   // Last mode code
      wStatusWord : Word;   // VFD Status word
      iActualSpeed : Int;   // VFD Actual speed
      wControlWord : Word;   // VFD Control word output
      iSpeedSetPoint : Int;   // VFD Speed output
      rCommandSpeed : Real;   // Speed command
      bNewMode : Bool;   // New mode selected
      bEnableForward : Bool;   // Forward enabled
      bEnableReverse : Bool;   // Reverse enabled
      bManualMode : Bool;   // Manual Mode is Active
      bAutoMode : Bool;   // Auto Mode is Active
      bRunTimeoutTimer : Bool;   // run the timeout timer
      bReset : Bool;
      bTON_TimeOut : Bool;
      bTON_ContactorDelay : Bool;
      bTON_CoolingFan : Bool;
      bTON_CurrentLimitDebounce : Bool;
      bPB_Forward : Bool;
      bPB_Reverse : Bool;
      bPB_Stop : Bool;
      bPB_ResetError : Bool;
   END_VAR
   VAR_TEMP
      CONTROL : Struct   // VFD Control Structure
         bON : Bool;   // On
         bOFF2 : Bool;   // Off2
         bOFF3 : Bool;   // Off3
         bENABLE_OPERATION : Bool;   // Enable Operation
         bDISABLE_RFG : Bool;   // Disable RFG
         bENABLE_RFG : Bool;   // Enable RFG
         bSETPOINT_ENABLE : Bool;   // Setpoint Enable
         bFAULT_ACK : Bool;   // Fault Acknowledge
         bCW_ACTIVATION : Bool;   // CW Activation
         bCCW_ACTIVATION : Bool;   // CCW Activation
         bSP_VALID : Bool;   // SP Valid
         bSP_INVERTED : Bool;   // SP Inverted
         bSPARE01 : Bool;   // Spare
         bMOTOR_POT_UP : Bool;   // Motor Pot up
         bMOTOR_POT_DN : Bool;   // Motor Pot down
         bLOCAL_ACTIVE : Bool;   // Local Active
      END_STRUCT;
      STATUS : Struct   // VFD Status Structure
         bAT_SETPOINT_FREQ : Bool;   // At Setpoint Frequency
         bMASTER_CONTROL : Bool;   // Master Control
         bMAX_FREQ_REACHED : Bool;   // Max Frequency Reached
         bCURRENT_LIMIT : Bool;   // Current Limit
         bBRAKE_ACTIVE : Bool;   // Brake Active
         bMOTOR_OVERLOAD : Bool;   // Motor Overload
         bCW_ROTATION : Bool;   // CW Rotation
         bINVERTER_OVERLOAD : Bool;   // Inverter Overload
         bREADY_FOR_ENABLE : Bool;   // Ready for Enable
         bREADY_TO_RUN : Bool;   // Ready To Run
         bRUNNING : Bool;   // Running
         bFAULT : Bool;   // Fault
         bOFF2_ACTIVE : Bool;   // Off2 Active
         bOFF3_ACTIVE : Bool;   // Off3 Active
         bSTART_LOCKOUT : Bool;   // Start Lockout
         bALARM : Bool;   // Alarm
      END_STRUCT;
      bMajorFault : Bool;   // Major Fault
      arrReadTemp : Array[1..6] of Word;
      dwWriteTemp : DWord;   // temporary dword
      bTemp : Bool;   // temp bit
      wTempWordValue : Word;   // used for temporaily holding a word value
      iTemp : Word;
      rTemp : Real;   // temporary real value
      tTemp : Time;   // temp time value
   END_VAR
   VAR CONSTANT
      crMaxSetPoint : Real := 200.0;   // Maximum speed set point
      crMinSetPoint : Real := 0.0;   // Minimum speed set point
      crSpeedScaling : Real := 163.84;   // Reference speed scale value
   END_VAR
   VAR_TEMP   // added for the SCL form of the ladder/FBD networks
      _w1 : Bool;
      _w2 : Bool;
      _w3 : Bool;
      _w4 : Bool;
   END_VAR
BEGIN

REGION Network 1: --------------------------------------------------------- Inputs ------------------------------------------------------------------
END_REGION

REGION Network 2: Read HMI input buttons
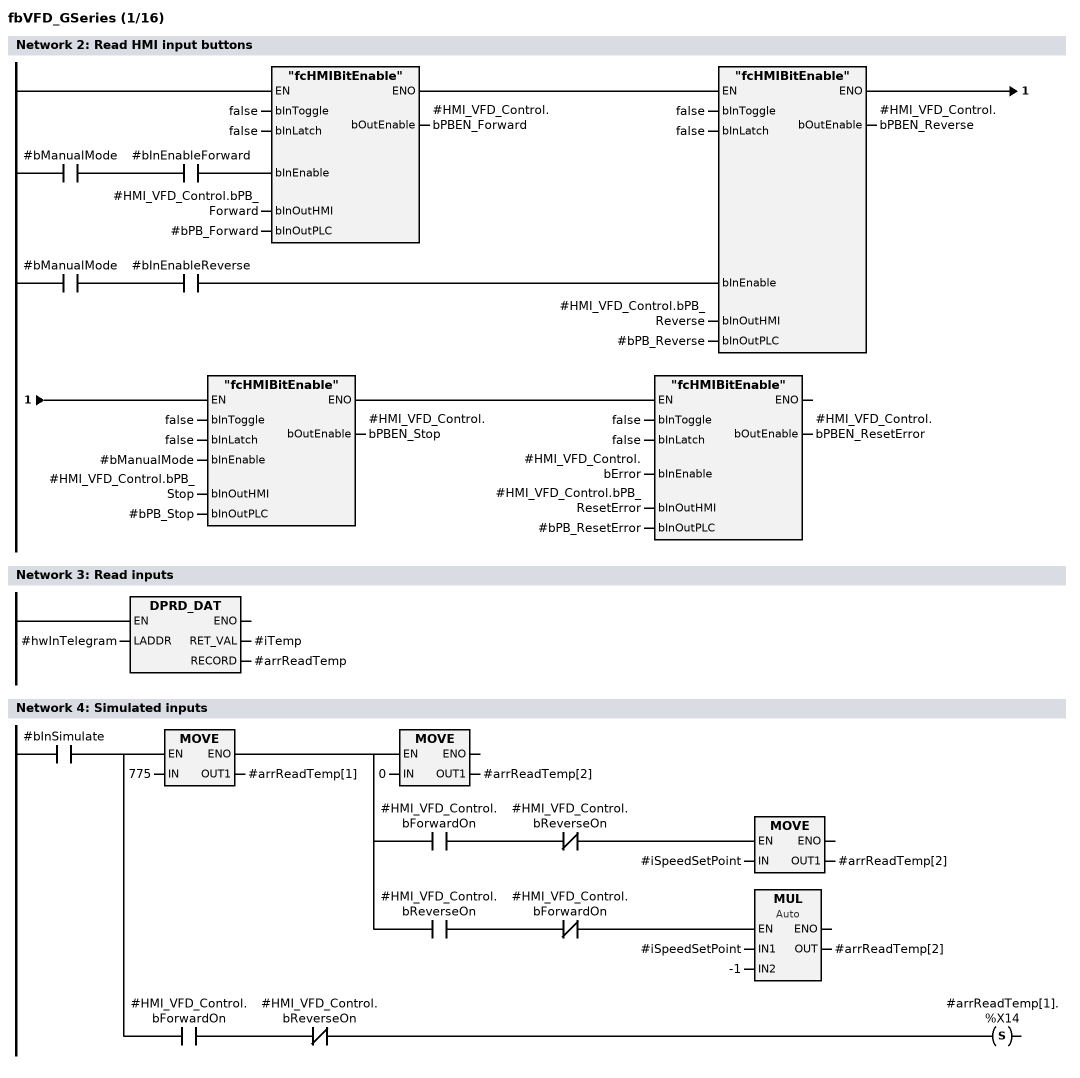
   RUNG wire#powerrail
      "fcHMIBitEnable"(bInEnable := wire#w1, bInToggle := false, bInLatch := false, bInOutHMI := #HMI_VFD_Control.bPB_Forward, bInOutPLC := #bPB_Forward, bOutEnable => #HMI_VFD_Control.bPBEN_Forward)
      "fcHMIBitEnable"(bInEnable := wire#w2, bInToggle := false, bInLatch := false, bInOutHMI := #HMI_VFD_Control.bPB_Reverse, bInOutPLC := #bPB_Reverse, bOutEnable => #HMI_VFD_Control.bPBEN_Reverse)
      "fcHMIBitEnable"(bInToggle := false, bInLatch := false, bInEnable := #bManualMode, bInOutHMI := #HMI_VFD_Control.bPB_Stop, bInOutPLC := #bPB_Stop, bOutEnable => #HMI_VFD_Control.bPBEN_Stop)
      "fcHMIBitEnable"(bInToggle := false, bInLatch := false, bInEnable := #HMI_VFD_Control.bError, bInOutHMI := #HMI_VFD_Control.bPB_ResetError, bInOutPLC := #bPB_ResetError, bOutEnable => #HMI_VFD_Control.bPBEN_ResetError)
   END_RUNG
   RUNG wire#powerrail
      Contact( #bManualMode )
      Contact( #bInEnableForward )
   END_RUNG wire#w1
   RUNG wire#powerrail
      Contact( #bManualMode )
      Contact( #bInEnableReverse )
   END_RUNG wire#w2
   // the same network as SCL:
   "fcHMIBitEnable"(bInToggle := false,
                    bInLatch := false,
                    bInEnable := #bManualMode AND #bInEnableForward,
                    bInOutHMI := #HMI_VFD_Control.bPB_Forward,
                    bInOutPLC := #bPB_Forward,
                    bOutEnable => #HMI_VFD_Control.bPBEN_Forward,
                    ENO => #_w1);
   "fcHMIBitEnable"(EN := #_w1,
                    bInToggle := false,
                    bInLatch := false,
                    bInEnable := #bManualMode AND #bInEnableReverse,
                    bInOutHMI := #HMI_VFD_Control.bPB_Reverse,
                    bInOutPLC := #bPB_Reverse,
                    bOutEnable => #HMI_VFD_Control.bPBEN_Reverse,
                    ENO => #_w2);
   "fcHMIBitEnable"(EN := #_w2,
                    bInToggle := false,
                    bInLatch := false,
                    bInEnable := #bManualMode,
                    bInOutHMI := #HMI_VFD_Control.bPB_Stop,
                    bInOutPLC := #bPB_Stop,
                    bOutEnable => #HMI_VFD_Control.bPBEN_Stop,
                    ENO => #_w3);
   IF #_w3 THEN
       "fcHMIBitEnable"(bInToggle := false,
                        bInLatch := false,
                        bInEnable := #HMI_VFD_Control.bError,
                        bInOutHMI := #HMI_VFD_Control.bPB_ResetError,
                        bInOutPLC := #bPB_ResetError,
                        bOutEnable => #HMI_VFD_Control.bPBEN_ResetError);
   END_IF;
END_REGION

REGION Network 3: Read inputs
   #iTemp := DPRD_DAT(LADDR := #hwInTelegram, RECORD => #arrReadTemp);
END_REGION

REGION Network 4: Simulated inputs
   RUNG wire#powerrail
      Contact( #bInSimulate )
      wire#w1
      Move(in := 775, out1 => #arrReadTemp[1])
      wire#w2
      Move(in := 0, out1 => #arrReadTemp[2])
   END_RUNG
   RUNG wire#w2
      Contact( #HMI_VFD_Control.bForwardOn )
      I_Contact( #HMI_VFD_Control.bReverseOn )
      Move(in := #iSpeedSetPoint, out1 => #arrReadTemp[2])
   END_RUNG
   RUNG wire#w2
      Contact( #HMI_VFD_Control.bReverseOn )
      I_Contact( #HMI_VFD_Control.bForwardOn )
      Mul(in1 := #iSpeedSetPoint, in2 := -1, out => #arrReadTemp[2])
   END_RUNG
   RUNG wire#w1
      Contact( #HMI_VFD_Control.bForwardOn )
      I_Contact( #HMI_VFD_Control.bReverseOn )
      S_Coil( #arrReadTemp[1].%X14 )
   END_RUNG
   // the same network as SCL:
   IF #bInSimulate THEN
       #arrReadTemp[1] := 775;
       #arrReadTemp[2] := 0;
   END_IF;
   IF #bInSimulate AND #HMI_VFD_Control.bForwardOn AND NOT #HMI_VFD_Control.bReverseOn THEN
       #arrReadTemp[2] := #iSpeedSetPoint;
   END_IF;
   IF #bInSimulate AND #HMI_VFD_Control.bReverseOn AND NOT #HMI_VFD_Control.bForwardOn THEN
       #arrReadTemp[2] := #iSpeedSetPoint * (-1);
   END_IF;
   IF #bInSimulate AND #HMI_VFD_Control.bForwardOn AND NOT #HMI_VFD_Control.bReverseOn THEN
       #arrReadTemp[1].%X14 := TRUE;
   END_IF;
END_REGION

REGION Network 5: Read the status word and parse to bits
   // // Read status word.  First word at iInAddress is the status word
   // wStatusWord := PIW[iInAddress];
   // 
   // fcWordToBits( wIN_WORD                    := wStatusWord,  // Parse status word
   //                 bOUT_BIT00                  := STATUS.bREADY_FOR_ENABLE,
   //                 bOUT_BIT01                  := STATUS.bREADY_TO_RUN,
   //                 bOUT_BIT02                  := STATUS.bRUNNING,
   //                 bOUT_BIT03                  := STATUS.bFAULT,
   //                 bOUT_BIT04                  := STATUS.bOFF2_ACTIVE,
   //                 bOUT_BIT05                  := STATUS.bOFF3_ACTIVE,
   //                 bOUT_BIT06                  := STATUS.bSTART_LOCKOUT,
   //                 bOUT_BIT07                  := STATUS.bALARM,
   //                 bOUT_BIT08                  := STATUS.bAT_SETPOINT_FREQ,
   //                 bOUT_BIT09                  := STATUS.bMASTER_CONTROL,
   //                 bOUT_BIT10                  := STATUS.bMAX_FREQ_REACHED,
   //                 bOUT_BIT11                  := STATUS.bCURRENT_LIMIT,
   //                 bOUT_BIT12                  := STATUS.bBRAKE_ACTIVE,
   //                 bOUT_BIT13                  := STATUS.bMOTOR_OVERLOAD,
   //                 bOUT_BIT14                  := STATUS.bCW_ROTATION,
   //                 bOUT_BIT15                  := STATUS.bINVERTER_OVERLOAD);
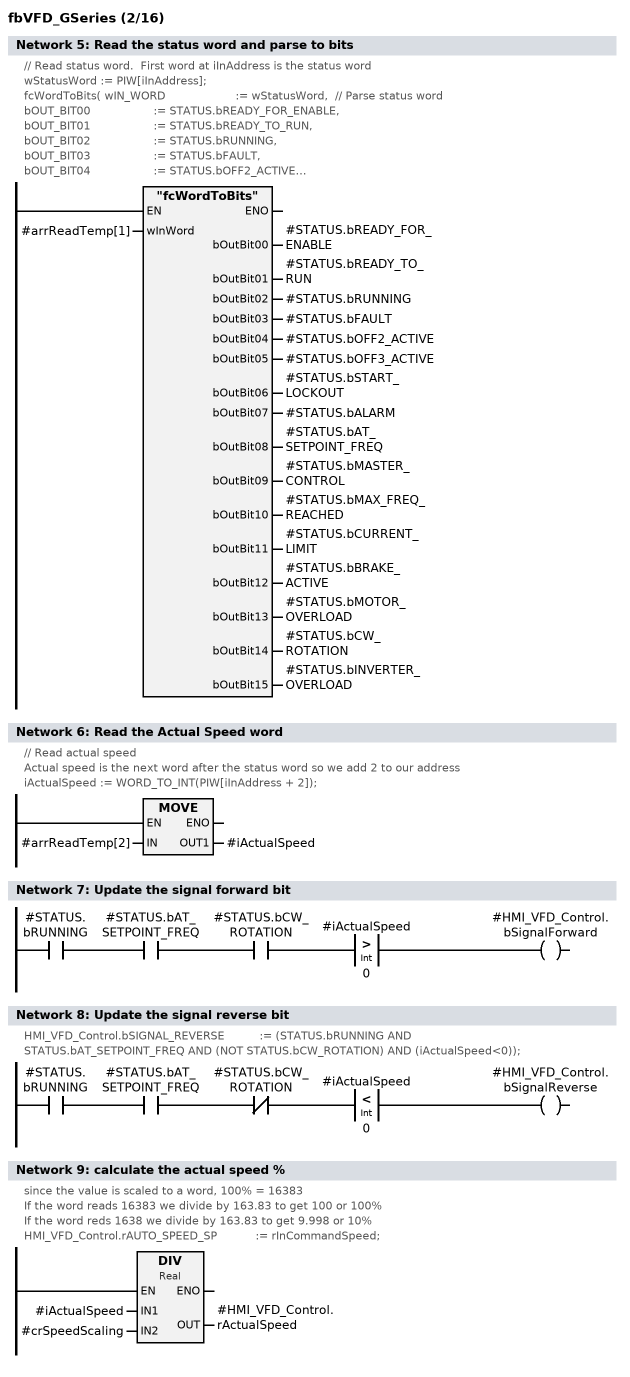
   RUNG wire#powerrail
      "fcWordToBits"(wInWord := #arrReadTemp[1], bOutBit00 => #STATUS.bREADY_FOR_ENABLE, bOutBit01 => #STATUS.bREADY_TO_RUN, bOutBit02 => #STATUS.bRUNNING, bOutBit03 => #STATUS.bFAULT, bOutBit04 => #STATUS.bOFF2_ACTIVE, bOutBit05 => #STATUS.bOFF3_ACTIVE, bOutBit06 => #STATUS.bSTART_LOCKOUT, bOutBit07 => #STATUS.bALARM, bOutBit08 => #STATUS.bAT_SETPOINT_FREQ, bOutBit09 => #STATUS.bMASTER_CONTROL, bOutBit10 => #STATUS.bMAX_FREQ_REACHED, bOutBit11 => #STATUS.bCURRENT_LIMIT, bOutBit12 => #STATUS.bBRAKE_ACTIVE, bOutBit13 => #STATUS.bMOTOR_OVERLOAD, bOutBit14 => #STATUS.bCW_ROTATION, bOutBit15 => #STATUS.bINVERTER_OVERLOAD)
   END_RUNG
   // the same network as SCL:
   "fcWordToBits"(wInWord := #arrReadTemp[1],
                  bOutBit00 => #STATUS.bREADY_FOR_ENABLE,
                  bOutBit01 => #STATUS.bREADY_TO_RUN,
                  bOutBit02 => #STATUS.bRUNNING,
                  bOutBit03 => #STATUS.bFAULT,
                  bOutBit04 => #STATUS.bOFF2_ACTIVE,
                  bOutBit05 => #STATUS.bOFF3_ACTIVE,
                  bOutBit06 => #STATUS.bSTART_LOCKOUT,
                  bOutBit07 => #STATUS.bALARM,
                  bOutBit08 => #STATUS.bAT_SETPOINT_FREQ,
                  bOutBit09 => #STATUS.bMASTER_CONTROL,
                  bOutBit10 => #STATUS.bMAX_FREQ_REACHED,
                  bOutBit11 => #STATUS.bCURRENT_LIMIT,
                  bOutBit12 => #STATUS.bBRAKE_ACTIVE,
                  bOutBit13 => #STATUS.bMOTOR_OVERLOAD,
                  bOutBit14 => #STATUS.bCW_ROTATION,
                  bOutBit15 => #STATUS.bINVERTER_OVERLOAD);
END_REGION

REGION Network 6: Read the Actual Speed word
   // // Read actual speed
   // Actual speed is the next word after the status word so we add 2 to our address
   // iActualSpeed := WORD_TO_INT(PIW[iInAddress + 2]);
   RUNG wire#powerrail
      Move(in := #arrReadTemp[2], out1 => #iActualSpeed)
   END_RUNG
   // the same network as SCL:
   #iActualSpeed := #arrReadTemp[2];
END_REGION

REGION Network 7: Update the signal forward bit
   RUNG wire#powerrail
      Contact( #STATUS.bRUNNING )
      Contact( #STATUS.bAT_SETPOINT_FREQ )
      Contact( #STATUS.bCW_ROTATION )
      { S7_Templates := "SrcType := Int" } GT_Contact(in1 := #iActualSpeed, in2 := 0)
      Coil( #HMI_VFD_Control.bSignalForward )
   END_RUNG
   // the same network as SCL:
   #HMI_VFD_Control.bSignalForward := #STATUS.bRUNNING AND #STATUS.bAT_SETPOINT_FREQ AND #STATUS.bCW_ROTATION AND (#iActualSpeed > 0);
END_REGION

REGION Network 8: Update the signal reverse bit
   // HMI_VFD_Control.bSIGNAL_REVERSE          := (STATUS.bRUNNING AND 
   // STATUS.bAT_SETPOINT_FREQ AND (NOT STATUS.bCW_ROTATION) AND (iActualSpeed<0));
   RUNG wire#powerrail
      Contact( #STATUS.bRUNNING )
      Contact( #STATUS.bAT_SETPOINT_FREQ )
      I_Contact( #STATUS.bCW_ROTATION )
      { S7_Templates := "SrcType := Int" } LT_Contact(in1 := #iActualSpeed, in2 := 0)
      Coil( #HMI_VFD_Control.bSignalReverse )
   END_RUNG
   // the same network as SCL:
   #HMI_VFD_Control.bSignalReverse := #STATUS.bRUNNING AND #STATUS.bAT_SETPOINT_FREQ AND NOT #STATUS.bCW_ROTATION AND (#iActualSpeed < 0);
END_REGION

REGION Network 9: calculate the actual speed %
   // since the value is scaled to a word, 100% = 16383
   // 
   // If the word reads 16383 we divide by 163.83 to get 100 or 100%
   // If the word reds 1638 we divide by 163.83 to get 9.998 or 10%
   // 
   // HMI_VFD_Control.rAUTO_SPEED_SP           := rInCommandSpeed;
   RUNG wire#powerrail
      { S7_Templates := "SrcType := Real" } Div(in1 := #iActualSpeed, in2 := #crSpeedScaling, out => #HMI_VFD_Control.rActualSpeed)
   END_RUNG
   // the same network as SCL:
   #HMI_VFD_Control.rActualSpeed := #iActualSpeed / #crSpeedScaling;
END_REGION

REGION Network 10: Set the automatic mode speed set point
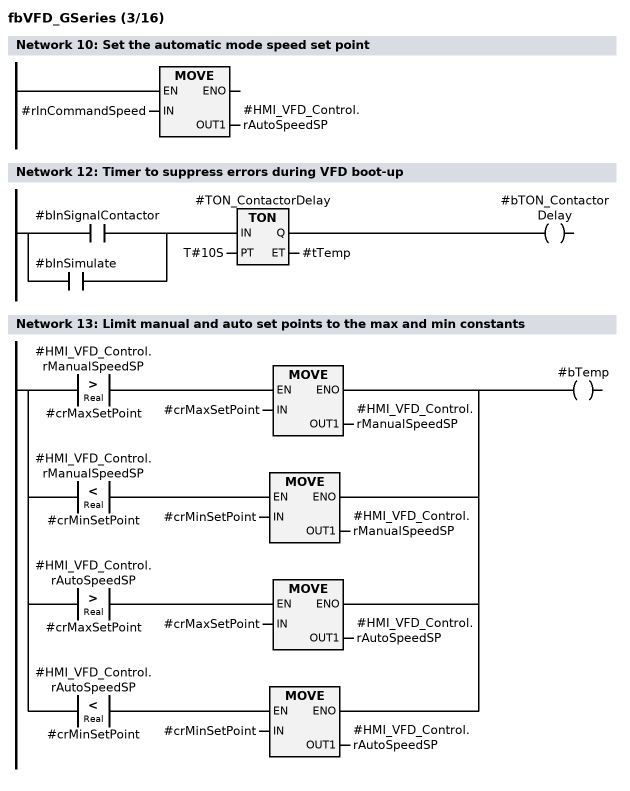
   RUNG wire#powerrail
      Move(in := #rInCommandSpeed, out1 => #HMI_VFD_Control.rAutoSpeedSP)
   END_RUNG
   // the same network as SCL:
   #HMI_VFD_Control.rAutoSpeedSP := #rInCommandSpeed;
END_REGION

REGION Network 11: --------------------------------------------------- Control Logic ------------------------------------------------------------
END_REGION

REGION Network 12: Timer to suppress errors during VFD boot-up
   #TON_ContactorDelay(IN := #bInSignalContactor OR #bInSimulate, PT := T#10S, ET => #tTemp);   // TON
   #bTON_ContactorDelay := #TON_ContactorDelay.Q;
END_REGION

REGION Network 13: Limit manual and auto set points to the max and min constants
   RUNG wire#powerrail
      { S7_Templates := "SrcType := Real" } GT_Contact(in1 := #HMI_VFD_Control.rManualSpeedSP, in2 := #crMaxSetPoint)
      Move(in := #crMaxSetPoint, out1 => #HMI_VFD_Control.rManualSpeedSP)
      wire#w1
      Coil( #bTemp )
   END_RUNG
   RUNG wire#powerrail
      { S7_Templates := "SrcType := Real" } LT_Contact(in1 := #HMI_VFD_Control.rManualSpeedSP, in2 := #crMinSetPoint)
      Move(in := #crMinSetPoint, out1 => #HMI_VFD_Control.rManualSpeedSP)
   END_RUNG wire#w1
   RUNG wire#powerrail
      { S7_Templates := "SrcType := Real" } GT_Contact(in1 := #HMI_VFD_Control.rAutoSpeedSP, in2 := #crMaxSetPoint)
      Move(in := #crMaxSetPoint, out1 => #HMI_VFD_Control.rAutoSpeedSP)
   END_RUNG wire#w1
   RUNG wire#powerrail
      { S7_Templates := "SrcType := Real" } LT_Contact(in1 := #HMI_VFD_Control.rAutoSpeedSP, in2 := #crMinSetPoint)
      Move(in := #crMinSetPoint, out1 => #HMI_VFD_Control.rAutoSpeedSP)
   END_RUNG wire#w1
   // the same network as SCL:
   #_w1 := #HMI_VFD_Control.rManualSpeedSP > #crMaxSetPoint;
   IF #_w1 THEN #HMI_VFD_Control.rManualSpeedSP := #crMaxSetPoint; END_IF;
   #_w2 := #HMI_VFD_Control.rManualSpeedSP < #crMinSetPoint;
   IF #_w2 THEN #HMI_VFD_Control.rManualSpeedSP := #crMinSetPoint; END_IF;
   #_w3 := #HMI_VFD_Control.rAutoSpeedSP > #crMaxSetPoint;
   IF #_w3 THEN #HMI_VFD_Control.rAutoSpeedSP := #crMaxSetPoint; END_IF;
   #_w4 := #HMI_VFD_Control.rAutoSpeedSP < #crMinSetPoint;
   IF #_w4 THEN #HMI_VFD_Control.rAutoSpeedSP := #crMinSetPoint; END_IF;
   #bTemp := #_w1 OR #_w2 OR #_w3 OR #_w4;
END_REGION

REGION Network 14: Reset errors
   // Clear all errors
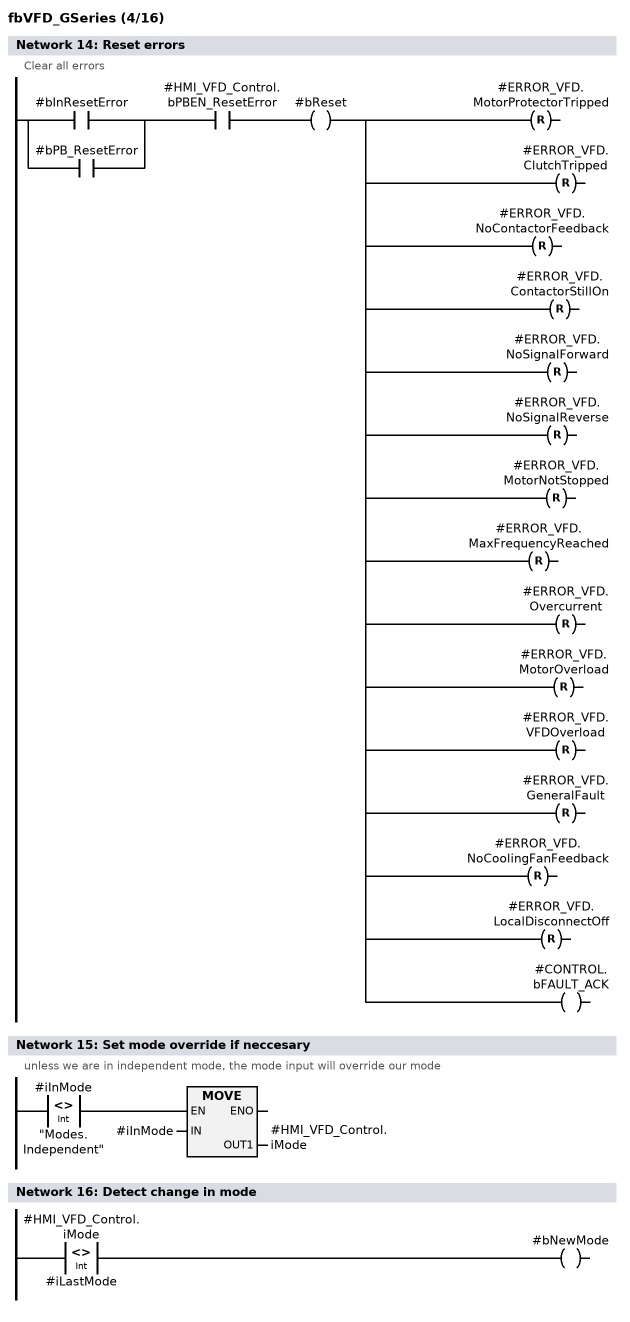
   RUNG wire#powerrail
      Contact( #bInResetError )
      wire#w1
      Contact( #HMI_VFD_Control.bPBEN_ResetError )
      Coil( #bReset )
      wire#w2
      R_Coil( #ERROR_VFD.MotorProtectorTripped )
   END_RUNG
   RUNG wire#powerrail
      Contact( #bPB_ResetError )
   END_RUNG wire#w1
   RUNG wire#w2
      R_Coil( #ERROR_VFD.ClutchTripped )
   END_RUNG
   RUNG wire#w2
      R_Coil( #ERROR_VFD.NoContactorFeedback )
   END_RUNG
   RUNG wire#w2
      R_Coil( #ERROR_VFD.ContactorStillOn )
   END_RUNG
   RUNG wire#w2
      R_Coil( #ERROR_VFD.NoSignalForward )
   END_RUNG
   RUNG wire#w2
      R_Coil( #ERROR_VFD.NoSignalReverse )
   END_RUNG
   RUNG wire#w2
      R_Coil( #ERROR_VFD.MotorNotStopped )
   END_RUNG
   RUNG wire#w2
      R_Coil( #ERROR_VFD.MaxFrequencyReached )
   END_RUNG
   RUNG wire#w2
      R_Coil( #ERROR_VFD.Overcurrent )
   END_RUNG
   RUNG wire#w2
      R_Coil( #ERROR_VFD.MotorOverload )
   END_RUNG
   RUNG wire#w2
      R_Coil( #ERROR_VFD.VFDOverload )
   END_RUNG
   RUNG wire#w2
      R_Coil( #ERROR_VFD.GeneralFault )
   END_RUNG
   RUNG wire#w2
      R_Coil( #ERROR_VFD.NoCoolingFanFeedback )
   END_RUNG
   RUNG wire#w2
      R_Coil( #ERROR_VFD.LocalDisconnectOff )
   END_RUNG
   RUNG wire#w2
      Coil( #CONTROL.bFAULT_ACK )
   END_RUNG
   // the same network as SCL:
   #bReset := (#bInResetError OR #bPB_ResetError) AND #HMI_VFD_Control.bPBEN_ResetError;
   IF #bReset THEN
       #ERROR_VFD.MotorProtectorTripped := FALSE;
       #ERROR_VFD.ClutchTripped := FALSE;
       #ERROR_VFD.NoContactorFeedback := FALSE;
       #ERROR_VFD.ContactorStillOn := FALSE;
       #ERROR_VFD.NoSignalForward := FALSE;
       #ERROR_VFD.NoSignalReverse := FALSE;
       #ERROR_VFD.MotorNotStopped := FALSE;
       #ERROR_VFD.MaxFrequencyReached := FALSE;
       #ERROR_VFD.Overcurrent := FALSE;
       #ERROR_VFD.MotorOverload := FALSE;
       #ERROR_VFD.VFDOverload := FALSE;
       #ERROR_VFD.GeneralFault := FALSE;
       #ERROR_VFD.NoCoolingFanFeedback := FALSE;
       #ERROR_VFD.LocalDisconnectOff := FALSE;
   END_IF;
   #CONTROL.bFAULT_ACK := #bReset;
END_REGION

REGION Network 15: Set mode override if neccesary
   // unless we are in independent mode, the mode input will override our mode
   RUNG wire#powerrail
      { S7_Templates := "SrcType := Int" } NE_Contact(in1 := #iInMode, in2 := "Modes.Independent")
      Move(in := #iInMode, out1 => #HMI_VFD_Control.iMode)
   END_RUNG
   // the same network as SCL:
   IF #iInMode <> "Modes.Independent" THEN #HMI_VFD_Control.iMode := #iInMode; END_IF;
END_REGION

REGION Network 16: Detect change in mode
   RUNG wire#powerrail
      { S7_Templates := "SrcType := Int" } NE_Contact(in1 := #HMI_VFD_Control.iMode, in2 := #iLastMode)
      Coil( #bNewMode )
   END_RUNG
   // the same network as SCL:
   #bNewMode := #HMI_VFD_Control.iMode <> #iLastMode;
END_REGION

REGION Network 17: Keep track of last mode
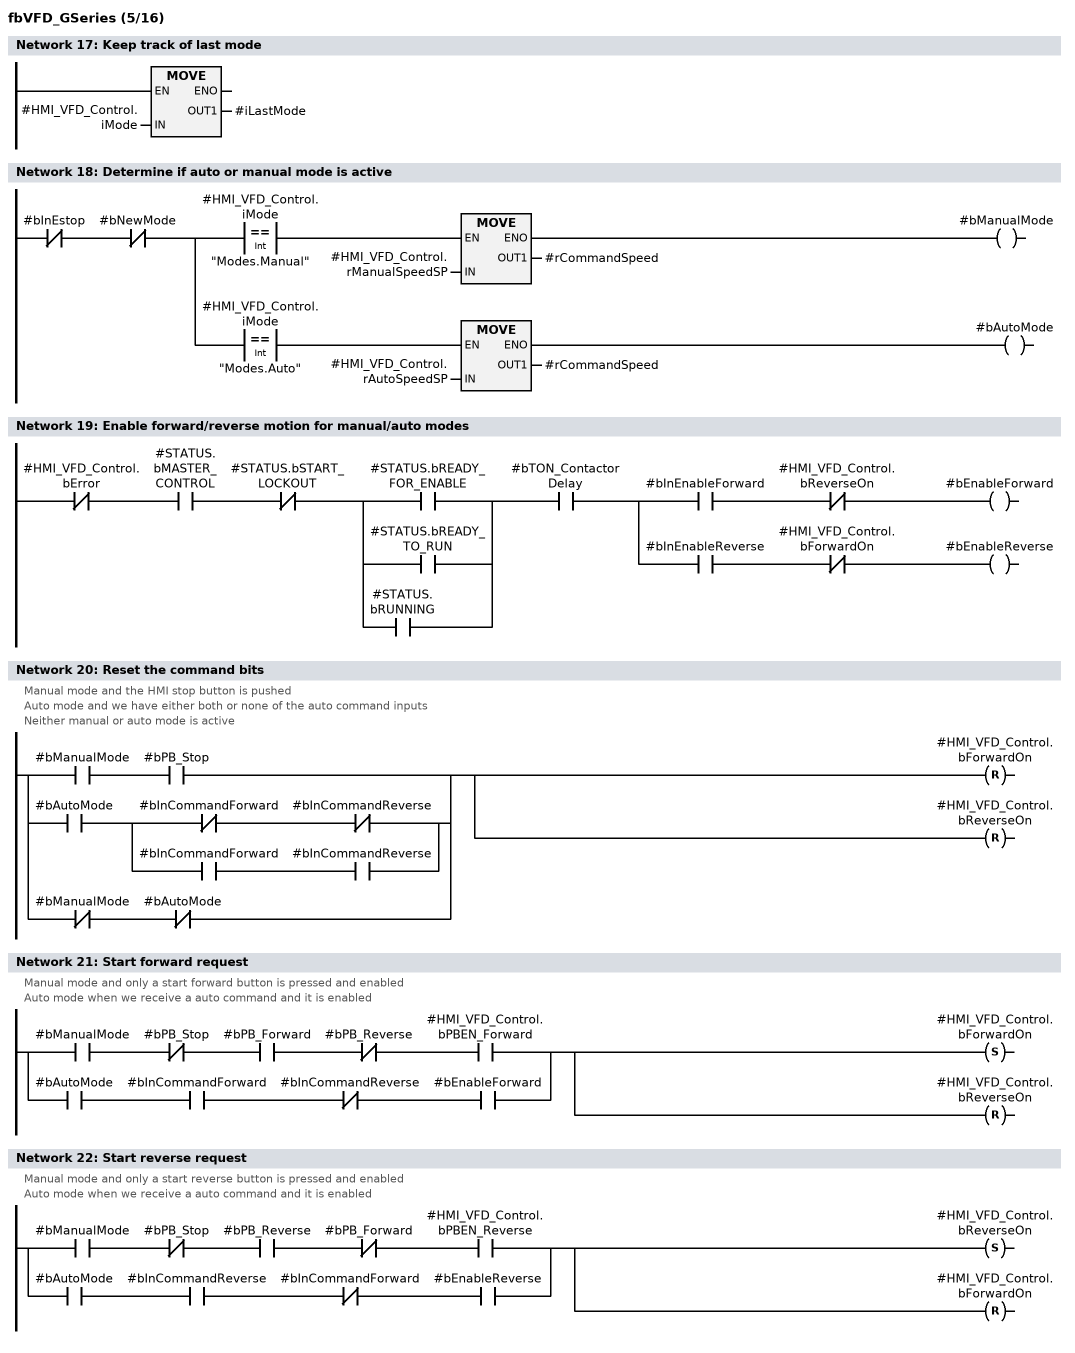
   RUNG wire#powerrail
      Move(in := #HMI_VFD_Control.iMode, out1 => #iLastMode)
   END_RUNG
   // the same network as SCL:
   #iLastMode := #HMI_VFD_Control.iMode;
END_REGION

REGION Network 18: Determine if auto or manual mode is active
   RUNG wire#powerrail
      I_Contact( #bInEstop )
      I_Contact( #bNewMode )
      wire#w1
      { S7_Templates := "SrcType := Int" } EQ_Contact(in1 := #HMI_VFD_Control.iMode, in2 := "Modes.Manual")
      Move(in := #HMI_VFD_Control.rManualSpeedSP, out1 => #rCommandSpeed)
      Coil( #bManualMode )
   END_RUNG
   RUNG wire#w1
      { S7_Templates := "SrcType := Int" } EQ_Contact(in1 := #HMI_VFD_Control.iMode, in2 := "Modes.Auto")
      Move(in := #HMI_VFD_Control.rAutoSpeedSP, out1 => #rCommandSpeed)
      Coil( #bAutoMode )
   END_RUNG
   // the same network as SCL:
   #_w1 := NOT #bInEstop AND NOT #bNewMode;
   #_w2 := #_w1 AND (#HMI_VFD_Control.iMode = "Modes.Manual");
   IF #_w2 THEN #rCommandSpeed := #HMI_VFD_Control.rManualSpeedSP; END_IF;
   #bManualMode := #_w2;
   #_w3 := #_w1 AND (#HMI_VFD_Control.iMode = "Modes.Auto");
   IF #_w3 THEN #rCommandSpeed := #HMI_VFD_Control.rAutoSpeedSP; END_IF;
   #bAutoMode := #_w3;
END_REGION

REGION Network 19: Enable forward/reverse motion for manual/auto modes
   RUNG wire#powerrail
      I_Contact( #HMI_VFD_Control.bError )
      Contact( #STATUS.bMASTER_CONTROL )
      I_Contact( #STATUS.bSTART_LOCKOUT )
      wire#w1
      Contact( #STATUS.bREADY_FOR_ENABLE )
      wire#w2
      Contact( #bTON_ContactorDelay )
      wire#w3
      Contact( #bInEnableForward )
      I_Contact( #HMI_VFD_Control.bReverseOn )
      Coil( #bEnableForward )
   END_RUNG
   RUNG wire#w1
      Contact( #STATUS.bREADY_TO_RUN )
   END_RUNG wire#w2
   RUNG wire#w1
      Contact( #STATUS.bRUNNING )
   END_RUNG wire#w2
   RUNG wire#w3
      Contact( #bInEnableReverse )
      I_Contact( #HMI_VFD_Control.bForwardOn )
      Coil( #bEnableReverse )
   END_RUNG
   // the same network as SCL:
   #_w1 := NOT #HMI_VFD_Control.bError AND #STATUS.bMASTER_CONTROL AND NOT #STATUS.bSTART_LOCKOUT AND (#STATUS.bREADY_FOR_ENABLE OR #STATUS.bREADY_TO_RUN OR #STATUS.bRUNNING) AND #bTON_ContactorDelay;
   #bEnableForward := #_w1 AND #bInEnableForward AND NOT #HMI_VFD_Control.bReverseOn;
   #bEnableReverse := #_w1 AND #bInEnableReverse AND NOT #HMI_VFD_Control.bForwardOn;
END_REGION

REGION Network 20: Reset the command bits
   // Manual mode and the HMI stop button is pushed
   // Auto mode and we have either both or none of the auto command inputs
   // Neither manual or auto mode is active
   RUNG wire#powerrail
      Contact( #bManualMode )
      Contact( #bPB_Stop )
      wire#w1
      R_Coil( #HMI_VFD_Control.bForwardOn )
   END_RUNG
   RUNG wire#powerrail
      Contact( #bAutoMode )
      wire#w2
      I_Contact( #bInCommandForward )
      I_Contact( #bInCommandReverse )
   END_RUNG wire#w1
   RUNG wire#w2
      Contact( #bInCommandForward )
      Contact( #bInCommandReverse )
   END_RUNG wire#w1
   RUNG wire#powerrail
      I_Contact( #bManualMode )
      I_Contact( #bAutoMode )
   END_RUNG wire#w1
   RUNG wire#w1
      R_Coil( #HMI_VFD_Control.bReverseOn )
   END_RUNG
   // the same network as SCL:
   IF (#bManualMode AND #bPB_Stop) OR (#bAutoMode AND ((NOT #bInCommandForward AND NOT #bInCommandReverse) OR (#bInCommandForward AND #bInCommandReverse))) OR (NOT #bManualMode AND NOT #bAutoMode) THEN
       #HMI_VFD_Control.bForwardOn := FALSE;
       #HMI_VFD_Control.bReverseOn := FALSE;
   END_IF;
END_REGION

REGION Network 21: Start forward request
   // Manual mode and only a start forward button is pressed and enabled
   // Auto mode when we receive a auto command and it is enabled
   RUNG wire#powerrail
      Contact( #bManualMode )
      I_Contact( #bPB_Stop )
      Contact( #bPB_Forward )
      I_Contact( #bPB_Reverse )
      Contact( #HMI_VFD_Control.bPBEN_Forward )
      wire#w1
      S_Coil( #HMI_VFD_Control.bForwardOn )
   END_RUNG
   RUNG wire#powerrail
      Contact( #bAutoMode )
      Contact( #bInCommandForward )
      I_Contact( #bInCommandReverse )
      Contact( #bEnableForward )
   END_RUNG wire#w1
   RUNG wire#w1
      R_Coil( #HMI_VFD_Control.bReverseOn )
   END_RUNG
   // the same network as SCL:
   IF (#bManualMode AND NOT #bPB_Stop AND #bPB_Forward AND NOT #bPB_Reverse AND #HMI_VFD_Control.bPBEN_Forward) OR (#bAutoMode AND #bInCommandForward AND NOT #bInCommandReverse AND #bEnableForward) THEN
       #HMI_VFD_Control.bForwardOn := TRUE;
       #HMI_VFD_Control.bReverseOn := FALSE;
   END_IF;
END_REGION

REGION Network 22: Start reverse request
   // Manual mode and only a start reverse button is pressed and enabled
   // Auto mode when we receive a auto command and it is enabled
   RUNG wire#powerrail
      Contact( #bManualMode )
      I_Contact( #bPB_Stop )
      Contact( #bPB_Reverse )
      I_Contact( #bPB_Forward )
      Contact( #HMI_VFD_Control.bPBEN_Reverse )
      wire#w1
      S_Coil( #HMI_VFD_Control.bReverseOn )
   END_RUNG
   RUNG wire#powerrail
      Contact( #bAutoMode )
      Contact( #bInCommandReverse )
      I_Contact( #bInCommandForward )
      Contact( #bEnableReverse )
   END_RUNG wire#w1
   RUNG wire#w1
      R_Coil( #HMI_VFD_Control.bForwardOn )
   END_RUNG
   // the same network as SCL:
   IF (#bManualMode AND NOT #bPB_Stop AND #bPB_Reverse AND NOT #bPB_Forward AND #HMI_VFD_Control.bPBEN_Reverse) OR (#bAutoMode AND #bInCommandReverse AND NOT #bInCommandForward AND #bEnableReverse) THEN
       #HMI_VFD_Control.bReverseOn := TRUE;
       #HMI_VFD_Control.bForwardOn := FALSE;
   END_IF;
END_REGION

REGION Network 23: If the forward enable is lost, stop the forward motion
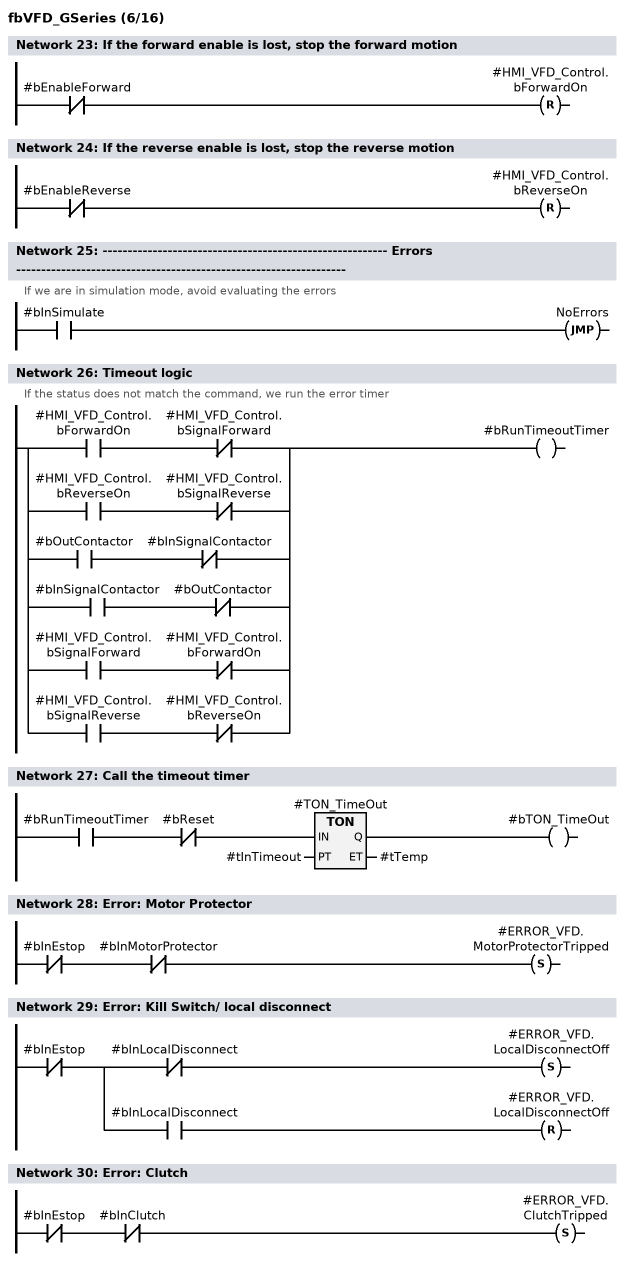
   RUNG wire#powerrail
      I_Contact( #bEnableForward )
      R_Coil( #HMI_VFD_Control.bForwardOn )
   END_RUNG
   // the same network as SCL:
   IF NOT #bEnableForward THEN #HMI_VFD_Control.bForwardOn := FALSE; END_IF;
END_REGION

REGION Network 24: If the reverse enable is lost, stop the reverse motion
   RUNG wire#powerrail
      I_Contact( #bEnableReverse )
      R_Coil( #HMI_VFD_Control.bReverseOn )
   END_RUNG
   // the same network as SCL:
   IF NOT #bEnableReverse THEN #HMI_VFD_Control.bReverseOn := FALSE; END_IF;
END_REGION

REGION Network 25: --------------------------------------------------------- Errors ------------------------------------------------------------------
   // If we are in simulation mode, avoid evaluating the errors
   RUNG wire#powerrail
      Contact( #bInSimulate )
      JumpCoil( NoErrors )
   END_RUNG
   // the same network as SCL:
   IF #bInSimulate THEN GOTO NoErrors; END_IF;
END_REGION

REGION Network 26: Timeout logic
   // If the status does not match the command, we run the error timer
   RUNG wire#powerrail
      Contact( #HMI_VFD_Control.bForwardOn )
      I_Contact( #HMI_VFD_Control.bSignalForward )
      wire#w1
      Coil( #bRunTimeoutTimer )
   END_RUNG
   RUNG wire#powerrail
      Contact( #HMI_VFD_Control.bReverseOn )
      I_Contact( #HMI_VFD_Control.bSignalReverse )
   END_RUNG wire#w1
   RUNG wire#powerrail
      Contact( #bOutContactor )
      I_Contact( #bInSignalContactor )
   END_RUNG wire#w1
   RUNG wire#powerrail
      Contact( #bInSignalContactor )
      I_Contact( #bOutContactor )
   END_RUNG wire#w1
   RUNG wire#powerrail
      Contact( #HMI_VFD_Control.bSignalForward )
      I_Contact( #HMI_VFD_Control.bForwardOn )
   END_RUNG wire#w1
   RUNG wire#powerrail
      Contact( #HMI_VFD_Control.bSignalReverse )
      I_Contact( #HMI_VFD_Control.bReverseOn )
   END_RUNG wire#w1
   // the same network as SCL:
   #bRunTimeoutTimer := (#HMI_VFD_Control.bForwardOn AND NOT #HMI_VFD_Control.bSignalForward) OR (#HMI_VFD_Control.bReverseOn AND NOT #HMI_VFD_Control.bSignalReverse) OR (#bOutContactor AND NOT #bInSignalContactor) OR (#bInSignalContactor AND NOT #bOutContactor) OR (#HMI_VFD_Control.bSignalForward AND NOT #HMI_VFD_Control.bForwardOn) OR (#HMI_VFD_Control.bSignalReverse AND NOT #HMI_VFD_Control.bReverseOn);
END_REGION

REGION Network 27: Call the timeout timer
   #TON_TimeOut(IN := #bRunTimeoutTimer AND NOT #bReset, PT := #tInTimeout, ET => #tTemp);   // TON
   #bTON_TimeOut := #TON_TimeOut.Q;
END_REGION

REGION Network 28: Error: Motor Protector
   RUNG wire#powerrail
      I_Contact( #bInEstop )
      I_Contact( #bInMotorProtector )
      S_Coil( #ERROR_VFD.MotorProtectorTripped )
   END_RUNG
   // the same network as SCL:
   IF NOT #bInEstop AND NOT #bInMotorProtector THEN #ERROR_VFD.MotorProtectorTripped := TRUE; END_IF;
END_REGION

REGION Network 29: Error: Kill Switch/ local disconnect
   RUNG wire#powerrail
      I_Contact( #bInEstop )
      wire#w1
      I_Contact( #bInLocalDisconnect )
      S_Coil( #ERROR_VFD.LocalDisconnectOff )
   END_RUNG
   RUNG wire#w1
      Contact( #bInLocalDisconnect )
      R_Coil( #ERROR_VFD.LocalDisconnectOff )
   END_RUNG
   // the same network as SCL:
   IF NOT #bInEstop AND NOT #bInLocalDisconnect THEN #ERROR_VFD.LocalDisconnectOff := TRUE; END_IF;
   IF NOT #bInEstop AND #bInLocalDisconnect THEN #ERROR_VFD.LocalDisconnectOff := FALSE; END_IF;
END_REGION

REGION Network 30: Error: Clutch
   RUNG wire#powerrail
      I_Contact( #bInEstop )
      I_Contact( #bInClutch )
      S_Coil( #ERROR_VFD.ClutchTripped )
   END_RUNG
   // the same network as SCL:
   IF NOT #bInEstop AND NOT #bInClutch THEN #ERROR_VFD.ClutchTripped := TRUE; END_IF;
END_REGION

REGION Network 31: Error: Max Frequency. This error isn't always used.
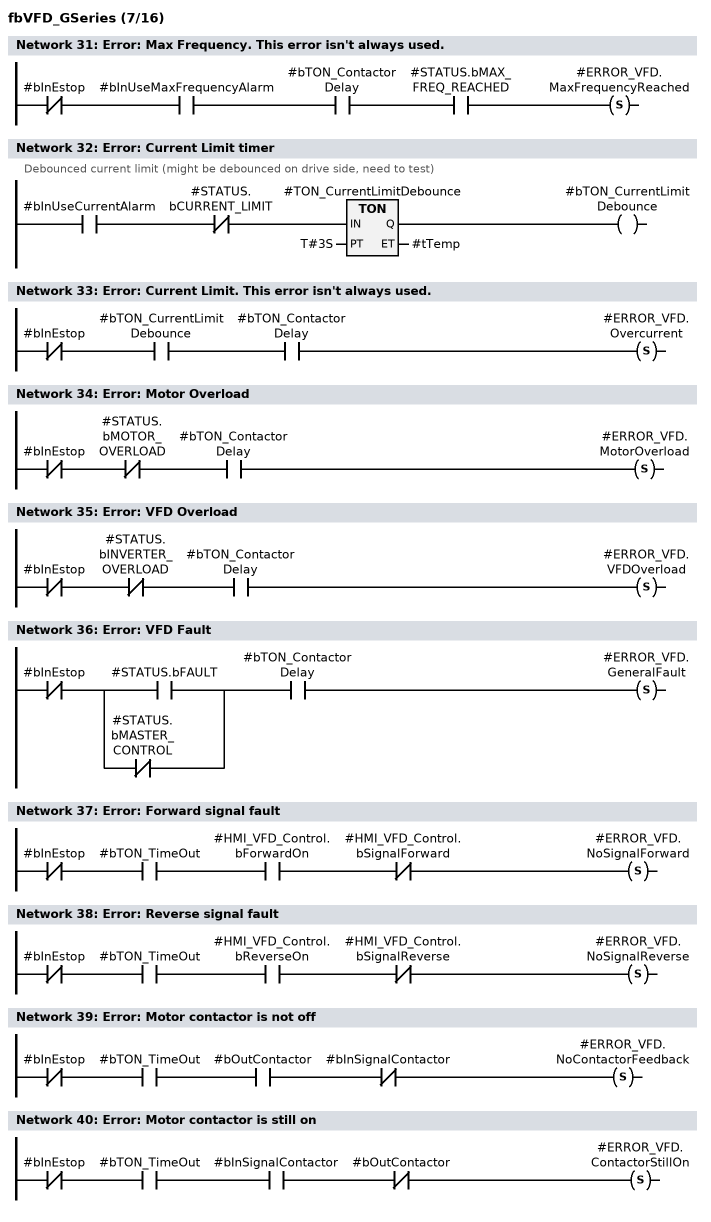
   RUNG wire#powerrail
      I_Contact( #bInEstop )
      Contact( #bInUseMaxFrequencyAlarm )
      Contact( #bTON_ContactorDelay )
      Contact( #STATUS.bMAX_FREQ_REACHED )
      S_Coil( #ERROR_VFD.MaxFrequencyReached )
   END_RUNG
   // the same network as SCL:
   IF NOT #bInEstop AND #bInUseMaxFrequencyAlarm AND #bTON_ContactorDelay AND #STATUS.bMAX_FREQ_REACHED THEN
       #ERROR_VFD.MaxFrequencyReached := TRUE;
   END_IF;
END_REGION

REGION Network 32: Error: Current Limit timer
   // Debounced current limit (might be debounced on drive side, need to test)
   #TON_CurrentLimitDebounce(IN := #bInUseCurrentAlarm AND NOT #STATUS.bCURRENT_LIMIT, PT := T#3S, ET => #tTemp);   // TON
   #bTON_CurrentLimitDebounce := #TON_CurrentLimitDebounce.Q;
END_REGION

REGION Network 33: Error: Current Limit. This error isn't always used.
   RUNG wire#powerrail
      I_Contact( #bInEstop )
      Contact( #bTON_CurrentLimitDebounce )
      Contact( #bTON_ContactorDelay )
      S_Coil( #ERROR_VFD.Overcurrent )
   END_RUNG
   // the same network as SCL:
   IF NOT #bInEstop AND #bTON_CurrentLimitDebounce AND #bTON_ContactorDelay THEN
       #ERROR_VFD.Overcurrent := TRUE;
   END_IF;
END_REGION

REGION Network 34: Error: Motor Overload
   RUNG wire#powerrail
      I_Contact( #bInEstop )
      I_Contact( #STATUS.bMOTOR_OVERLOAD )
      Contact( #bTON_ContactorDelay )
      S_Coil( #ERROR_VFD.MotorOverload )
   END_RUNG
   // the same network as SCL:
   IF NOT #bInEstop AND NOT #STATUS.bMOTOR_OVERLOAD AND #bTON_ContactorDelay THEN
       #ERROR_VFD.MotorOverload := TRUE;
   END_IF;
END_REGION

REGION Network 35: Error: VFD Overload
   RUNG wire#powerrail
      I_Contact( #bInEstop )
      I_Contact( #STATUS.bINVERTER_OVERLOAD )
      Contact( #bTON_ContactorDelay )
      S_Coil( #ERROR_VFD.VFDOverload )
   END_RUNG
   // the same network as SCL:
   IF NOT #bInEstop AND NOT #STATUS.bINVERTER_OVERLOAD AND #bTON_ContactorDelay THEN
       #ERROR_VFD.VFDOverload := TRUE;
   END_IF;
END_REGION

REGION Network 36: Error: VFD Fault
   RUNG wire#powerrail
      I_Contact( #bInEstop )
      wire#w1
      Contact( #STATUS.bFAULT )
      wire#w2
      Contact( #bTON_ContactorDelay )
      S_Coil( #ERROR_VFD.GeneralFault )
   END_RUNG
   RUNG wire#w1
      I_Contact( #STATUS.bMASTER_CONTROL )
   END_RUNG wire#w2
   // the same network as SCL:
   IF NOT #bInEstop AND (#STATUS.bFAULT OR NOT #STATUS.bMASTER_CONTROL) AND #bTON_ContactorDelay THEN
       #ERROR_VFD.GeneralFault := TRUE;
   END_IF;
END_REGION

REGION Network 37: Error: Forward signal fault
   RUNG wire#powerrail
      I_Contact( #bInEstop )
      Contact( #bTON_TimeOut )
      Contact( #HMI_VFD_Control.bForwardOn )
      I_Contact( #HMI_VFD_Control.bSignalForward )
      S_Coil( #ERROR_VFD.NoSignalForward )
   END_RUNG
   // the same network as SCL:
   IF NOT #bInEstop AND #bTON_TimeOut AND #HMI_VFD_Control.bForwardOn AND NOT #HMI_VFD_Control.bSignalForward THEN
       #ERROR_VFD.NoSignalForward := TRUE;
   END_IF;
END_REGION

REGION Network 38: Error: Reverse signal fault
   RUNG wire#powerrail
      I_Contact( #bInEstop )
      Contact( #bTON_TimeOut )
      Contact( #HMI_VFD_Control.bReverseOn )
      I_Contact( #HMI_VFD_Control.bSignalReverse )
      S_Coil( #ERROR_VFD.NoSignalReverse )
   END_RUNG
   // the same network as SCL:
   IF NOT #bInEstop AND #bTON_TimeOut AND #HMI_VFD_Control.bReverseOn AND NOT #HMI_VFD_Control.bSignalReverse THEN
       #ERROR_VFD.NoSignalReverse := TRUE;
   END_IF;
END_REGION

REGION Network 39: Error: Motor contactor is not off
   RUNG wire#powerrail
      I_Contact( #bInEstop )
      Contact( #bTON_TimeOut )
      Contact( #bOutContactor )
      I_Contact( #bInSignalContactor )
      S_Coil( #ERROR_VFD.NoContactorFeedback )
   END_RUNG
   // the same network as SCL:
   IF NOT #bInEstop AND #bTON_TimeOut AND #bOutContactor AND NOT #bInSignalContactor THEN
       #ERROR_VFD.NoContactorFeedback := TRUE;
   END_IF;
END_REGION

REGION Network 40: Error: Motor contactor is still on
   RUNG wire#powerrail
      I_Contact( #bInEstop )
      Contact( #bTON_TimeOut )
      Contact( #bInSignalContactor )
      I_Contact( #bOutContactor )
      S_Coil( #ERROR_VFD.ContactorStillOn )
   END_RUNG
   // the same network as SCL:
   IF NOT #bInEstop AND #bTON_TimeOut AND #bInSignalContactor AND NOT #bOutContactor THEN
       #ERROR_VFD.ContactorStillOn := TRUE;
   END_IF;
END_REGION

REGION Network 41: Error: Motor Doesn't stop
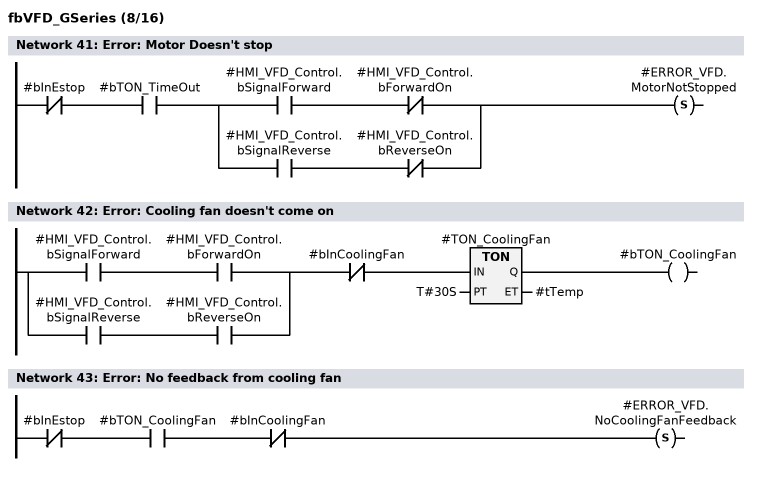
   RUNG wire#powerrail
      I_Contact( #bInEstop )
      Contact( #bTON_TimeOut )
      wire#w1
      Contact( #HMI_VFD_Control.bSignalForward )
      I_Contact( #HMI_VFD_Control.bForwardOn )
      wire#w2
      S_Coil( #ERROR_VFD.MotorNotStopped )
   END_RUNG
   RUNG wire#w1
      Contact( #HMI_VFD_Control.bSignalReverse )
      I_Contact( #HMI_VFD_Control.bReverseOn )
   END_RUNG wire#w2
   // the same network as SCL:
   IF NOT #bInEstop AND #bTON_TimeOut AND ((#HMI_VFD_Control.bSignalForward AND NOT #HMI_VFD_Control.bForwardOn) OR (#HMI_VFD_Control.bSignalReverse AND NOT #HMI_VFD_Control.bReverseOn)) THEN
       #ERROR_VFD.MotorNotStopped := TRUE;
   END_IF;
END_REGION

REGION Network 42: Error: Cooling fan doesn't come on
   #TON_CoolingFan(IN := ((#HMI_VFD_Control.bSignalForward AND #HMI_VFD_Control.bForwardOn) OR (#HMI_VFD_Control.bSignalReverse AND #HMI_VFD_Control.bReverseOn)) AND NOT #bInCoolingFan,   // TON
                   PT := T#30S,
                   ET => #tTemp);
   #bTON_CoolingFan := #TON_CoolingFan.Q;
END_REGION

REGION Network 43: Error: No feedback from cooling fan
   RUNG wire#powerrail
      I_Contact( #bInEstop )
      Contact( #bTON_CoolingFan )
      I_Contact( #bInCoolingFan )
      S_Coil( #ERROR_VFD.NoCoolingFanFeedback )
   END_RUNG
   // the same network as SCL:
   IF NOT #bInEstop AND #bTON_CoolingFan AND NOT #bInCoolingFan THEN
       #ERROR_VFD.NoCoolingFanFeedback := TRUE;
   END_IF;
END_REGION

REGION Network 44: Scroll errors on the HMI
   // Call the Error-Scroller which cyles through all possible errors and checks 
   // their state for display on the HMI
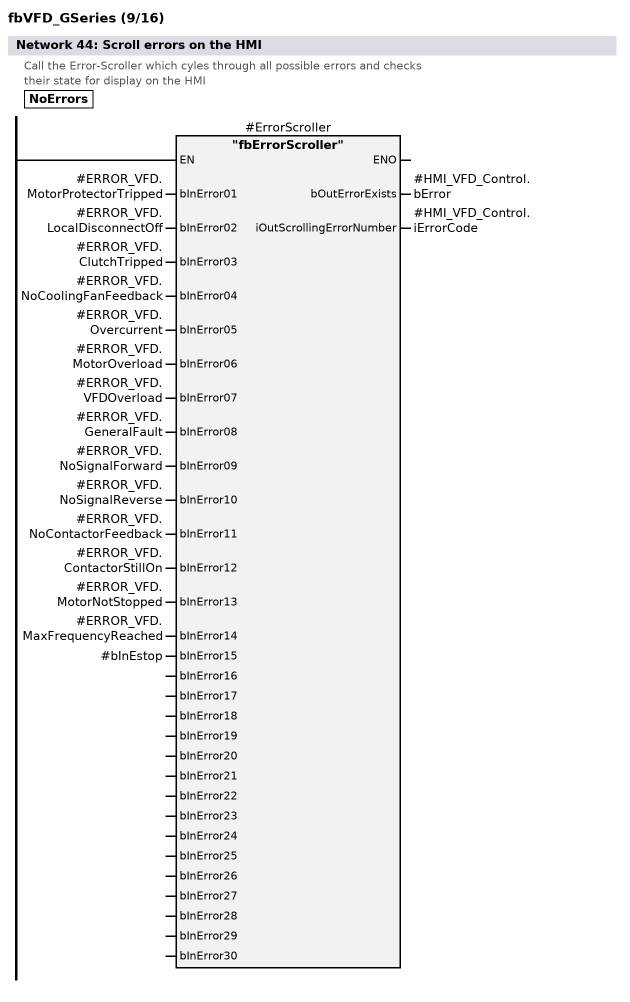
   Label( NoErrors )
   RUNG wire#powerrail
      #ErrorScroller(bInError01 := #ERROR_VFD.MotorProtectorTripped, bInError02 := #ERROR_VFD.LocalDisconnectOff, bInError03 := #ERROR_VFD.ClutchTripped, bInError04 := #ERROR_VFD.NoCoolingFanFeedback, bInError05 := #ERROR_VFD.Overcurrent, bInError06 := #ERROR_VFD.MotorOverload, bInError07 := #ERROR_VFD.VFDOverload, bInError08 := #ERROR_VFD.GeneralFault, bInError09 := #ERROR_VFD.NoSignalForward, bInError10 := #ERROR_VFD.NoSignalReverse, bInError11 := #ERROR_VFD.NoContactorFeedback, bInError12 := #ERROR_VFD.ContactorStillOn, bInError13 := #ERROR_VFD.MotorNotStopped, bInError14 := #ERROR_VFD.MaxFrequencyReached, bInError15 := #bInEstop, bInError16 :=, bInError17 :=, bInError18 :=, bInError19 :=, bInError20 :=, bInError21 :=, bInError22 :=, bInError23 :=, bInError24 :=, bInError25 :=, bInError26 :=, bInError27 :=, bInError28 :=, bInError29 :=, bInError30 :=, bOutErrorExists => #HMI_VFD_Control.bError, iOutScrollingErrorNumber => #HMI_VFD_Control.iErrorCode)
   END_RUNG
   // the same network as SCL:
   NoErrors:
   #ErrorScroller(bInError01 := #ERROR_VFD.MotorProtectorTripped,   // "fbErrorScroller"
                  bInError02 := #ERROR_VFD.LocalDisconnectOff,
                  bInError03 := #ERROR_VFD.ClutchTripped,
                  bInError04 := #ERROR_VFD.NoCoolingFanFeedback,
                  bInError05 := #ERROR_VFD.Overcurrent,
                  bInError06 := #ERROR_VFD.MotorOverload,
                  bInError07 := #ERROR_VFD.VFDOverload,
                  bInError08 := #ERROR_VFD.GeneralFault,
                  bInError09 := #ERROR_VFD.NoSignalForward,
                  bInError10 := #ERROR_VFD.NoSignalReverse,
                  bInError11 := #ERROR_VFD.NoContactorFeedback,
                  bInError12 := #ERROR_VFD.ContactorStillOn,
                  bInError13 := #ERROR_VFD.MotorNotStopped,
                  bInError14 := #ERROR_VFD.MaxFrequencyReached,
                  bInError15 := #bInEstop,
                  bOutErrorExists => #HMI_VFD_Control.bError,
                  iOutScrollingErrorNumber => #HMI_VFD_Control.iErrorCode);
END_REGION

REGION Network 45: Set major fault bit
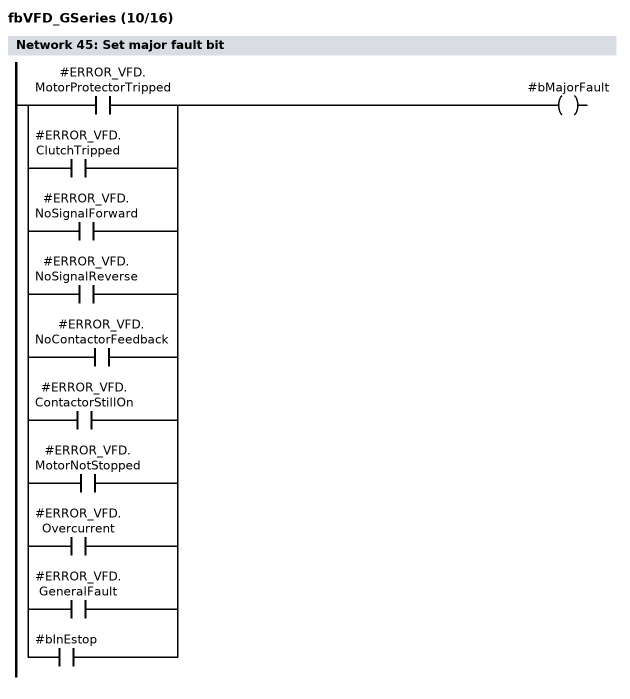
   RUNG wire#powerrail
      Contact( #ERROR_VFD.MotorProtectorTripped )
      wire#w1
      Coil( #bMajorFault )
   END_RUNG
   RUNG wire#powerrail
      Contact( #ERROR_VFD.ClutchTripped )
   END_RUNG wire#w1
   RUNG wire#powerrail
      Contact( #ERROR_VFD.NoSignalForward )
   END_RUNG wire#w1
   RUNG wire#powerrail
      Contact( #ERROR_VFD.NoSignalReverse )
   END_RUNG wire#w1
   RUNG wire#powerrail
      Contact( #ERROR_VFD.NoContactorFeedback )
   END_RUNG wire#w1
   RUNG wire#powerrail
      Contact( #ERROR_VFD.ContactorStillOn )
   END_RUNG wire#w1
   RUNG wire#powerrail
      Contact( #ERROR_VFD.MotorNotStopped )
   END_RUNG wire#w1
   RUNG wire#powerrail
      Contact( #ERROR_VFD.Overcurrent )
   END_RUNG wire#w1
   RUNG wire#powerrail
      Contact( #ERROR_VFD.GeneralFault )
   END_RUNG wire#w1
   RUNG wire#powerrail
      Contact( #bInEstop )
   END_RUNG wire#w1
   // the same network as SCL:
   #bMajorFault := #ERROR_VFD.MotorProtectorTripped OR #ERROR_VFD.ClutchTripped OR #ERROR_VFD.NoSignalForward OR #ERROR_VFD.NoSignalReverse OR #ERROR_VFD.NoContactorFeedback OR #ERROR_VFD.ContactorStillOn OR #ERROR_VFD.MotorNotStopped OR #ERROR_VFD.Overcurrent OR #ERROR_VFD.GeneralFault OR #bInEstop;
END_REGION

REGION Network 46: Set control bits based on major fault
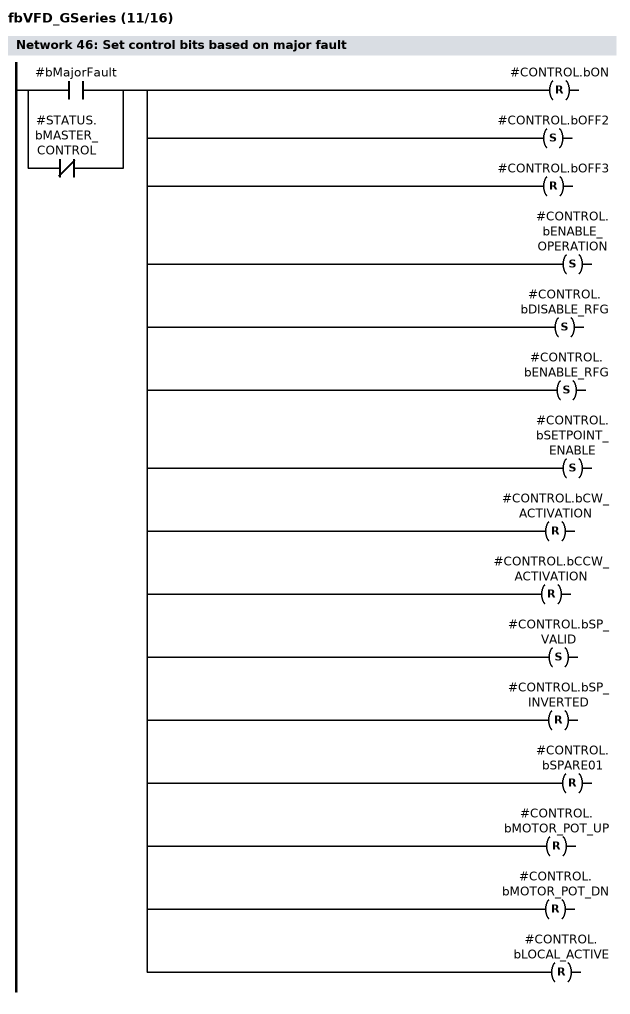
   RUNG wire#powerrail
      Contact( #bMajorFault )
      wire#w1
      R_Coil( #CONTROL.bON )
   END_RUNG
   RUNG wire#powerrail
      I_Contact( #STATUS.bMASTER_CONTROL )
   END_RUNG wire#w1
   RUNG wire#w1
      S_Coil( #CONTROL.bOFF2 )
   END_RUNG
   RUNG wire#w1
      R_Coil( #CONTROL.bOFF3 )
   END_RUNG
   RUNG wire#w1
      S_Coil( #CONTROL.bENABLE_OPERATION )
   END_RUNG
   RUNG wire#w1
      S_Coil( #CONTROL.bDISABLE_RFG )
   END_RUNG
   RUNG wire#w1
      S_Coil( #CONTROL.bENABLE_RFG )
   END_RUNG
   RUNG wire#w1
      S_Coil( #CONTROL.bSETPOINT_ENABLE )
   END_RUNG
   RUNG wire#w1
      R_Coil( #CONTROL.bCW_ACTIVATION )
   END_RUNG
   RUNG wire#w1
      R_Coil( #CONTROL.bCCW_ACTIVATION )
   END_RUNG
   RUNG wire#w1
      S_Coil( #CONTROL.bSP_VALID )
   END_RUNG
   RUNG wire#w1
      R_Coil( #CONTROL.bSP_INVERTED )
   END_RUNG
   RUNG wire#w1
      R_Coil( #CONTROL.bSPARE01 )
   END_RUNG
   RUNG wire#w1
      R_Coil( #CONTROL.bMOTOR_POT_UP )
   END_RUNG
   RUNG wire#w1
      R_Coil( #CONTROL.bMOTOR_POT_DN )
   END_RUNG
   RUNG wire#w1
      R_Coil( #CONTROL.bLOCAL_ACTIVE )
   END_RUNG
   // the same network as SCL:
   IF #bMajorFault OR NOT #STATUS.bMASTER_CONTROL THEN
       #CONTROL.bON := FALSE;
       #CONTROL.bOFF2 := TRUE;
       #CONTROL.bOFF3 := FALSE;
       #CONTROL.bENABLE_OPERATION := TRUE;
       #CONTROL.bDISABLE_RFG := TRUE;
       #CONTROL.bENABLE_RFG := TRUE;
       #CONTROL.bSETPOINT_ENABLE := TRUE;
       #CONTROL.bCW_ACTIVATION := FALSE;
       #CONTROL.bCCW_ACTIVATION := FALSE;
       #CONTROL.bSP_VALID := TRUE;
       #CONTROL.bSP_INVERTED := FALSE;
       #CONTROL.bSPARE01 := FALSE;
       #CONTROL.bMOTOR_POT_UP := FALSE;
       #CONTROL.bMOTOR_POT_DN := FALSE;
       #CONTROL.bLOCAL_ACTIVE := FALSE;
   END_IF;
END_REGION

REGION Network 47: Set control bits based on forward on command
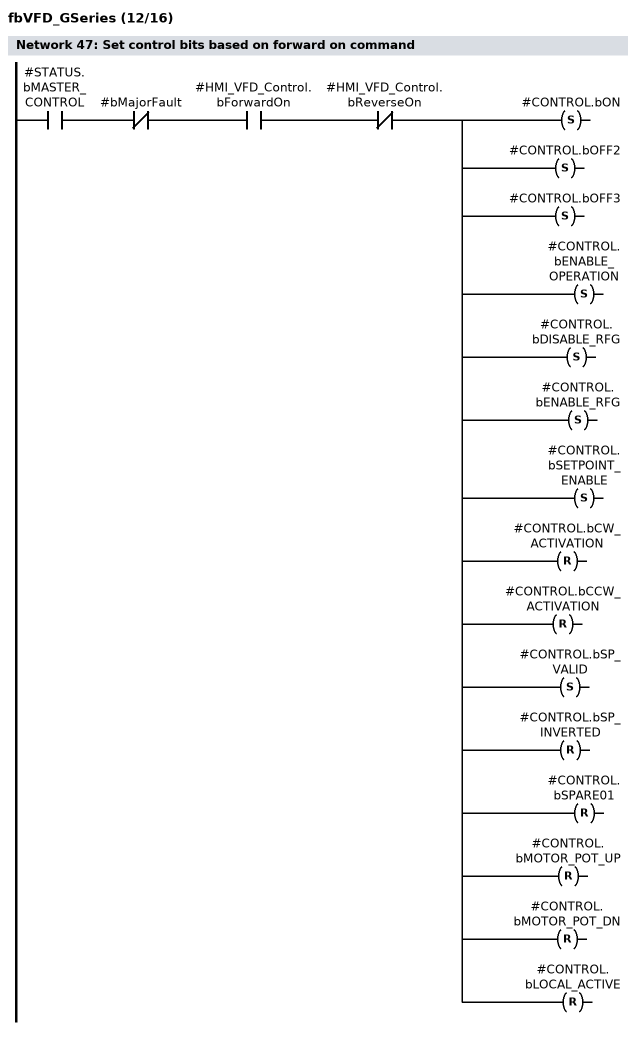
   RUNG wire#powerrail
      Contact( #STATUS.bMASTER_CONTROL )
      I_Contact( #bMajorFault )
      Contact( #HMI_VFD_Control.bForwardOn )
      I_Contact( #HMI_VFD_Control.bReverseOn )
      wire#w1
      S_Coil( #CONTROL.bON )
   END_RUNG
   RUNG wire#w1
      S_Coil( #CONTROL.bOFF2 )
   END_RUNG
   RUNG wire#w1
      S_Coil( #CONTROL.bOFF3 )
   END_RUNG
   RUNG wire#w1
      S_Coil( #CONTROL.bENABLE_OPERATION )
   END_RUNG
   RUNG wire#w1
      S_Coil( #CONTROL.bDISABLE_RFG )
   END_RUNG
   RUNG wire#w1
      S_Coil( #CONTROL.bENABLE_RFG )
   END_RUNG
   RUNG wire#w1
      S_Coil( #CONTROL.bSETPOINT_ENABLE )
   END_RUNG
   RUNG wire#w1
      R_Coil( #CONTROL.bCW_ACTIVATION )
   END_RUNG
   RUNG wire#w1
      R_Coil( #CONTROL.bCCW_ACTIVATION )
   END_RUNG
   RUNG wire#w1
      S_Coil( #CONTROL.bSP_VALID )
   END_RUNG
   RUNG wire#w1
      R_Coil( #CONTROL.bSP_INVERTED )
   END_RUNG
   RUNG wire#w1
      R_Coil( #CONTROL.bSPARE01 )
   END_RUNG
   RUNG wire#w1
      R_Coil( #CONTROL.bMOTOR_POT_UP )
   END_RUNG
   RUNG wire#w1
      R_Coil( #CONTROL.bMOTOR_POT_DN )
   END_RUNG
   RUNG wire#w1
      R_Coil( #CONTROL.bLOCAL_ACTIVE )
   END_RUNG
   // the same network as SCL:
   IF #STATUS.bMASTER_CONTROL AND NOT #bMajorFault AND #HMI_VFD_Control.bForwardOn AND NOT #HMI_VFD_Control.bReverseOn THEN
       #CONTROL.bON := TRUE;
       #CONTROL.bOFF2 := TRUE;
       #CONTROL.bOFF3 := TRUE;
       #CONTROL.bENABLE_OPERATION := TRUE;
       #CONTROL.bDISABLE_RFG := TRUE;
       #CONTROL.bENABLE_RFG := TRUE;
       #CONTROL.bSETPOINT_ENABLE := TRUE;
       #CONTROL.bCW_ACTIVATION := FALSE;
       #CONTROL.bCCW_ACTIVATION := FALSE;
       #CONTROL.bSP_VALID := TRUE;
       #CONTROL.bSP_INVERTED := FALSE;
       #CONTROL.bSPARE01 := FALSE;
       #CONTROL.bMOTOR_POT_UP := FALSE;
       #CONTROL.bMOTOR_POT_DN := FALSE;
       #CONTROL.bLOCAL_ACTIVE := FALSE;
   END_IF;
END_REGION

REGION Network 48: Set control bits based on Reverse on command
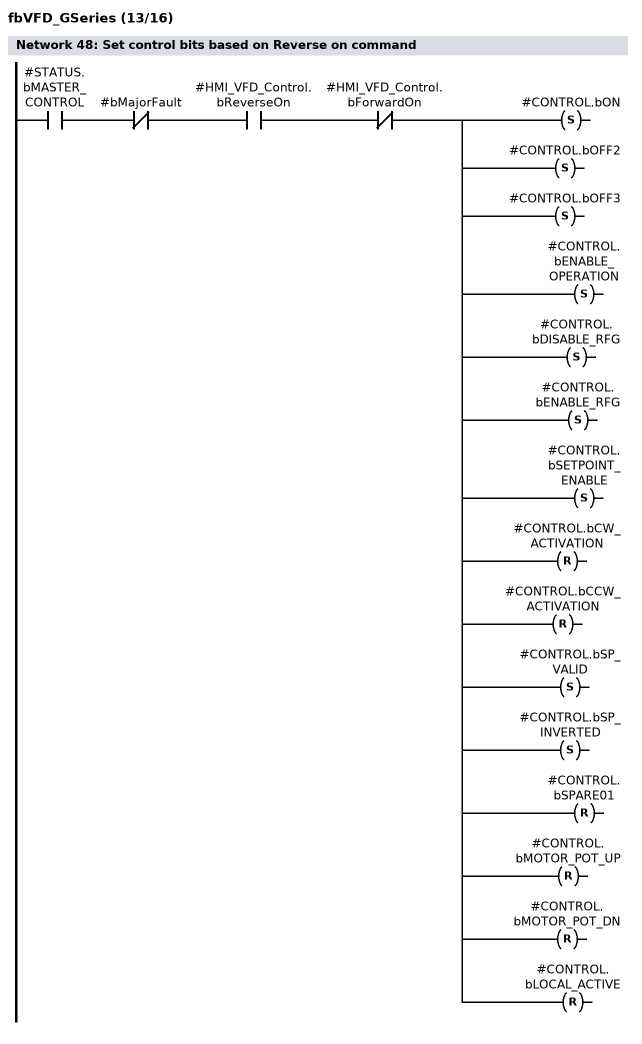
   RUNG wire#powerrail
      Contact( #STATUS.bMASTER_CONTROL )
      I_Contact( #bMajorFault )
      Contact( #HMI_VFD_Control.bReverseOn )
      I_Contact( #HMI_VFD_Control.bForwardOn )
      wire#w1
      S_Coil( #CONTROL.bON )
   END_RUNG
   RUNG wire#w1
      S_Coil( #CONTROL.bOFF2 )
   END_RUNG
   RUNG wire#w1
      S_Coil( #CONTROL.bOFF3 )
   END_RUNG
   RUNG wire#w1
      S_Coil( #CONTROL.bENABLE_OPERATION )
   END_RUNG
   RUNG wire#w1
      S_Coil( #CONTROL.bDISABLE_RFG )
   END_RUNG
   RUNG wire#w1
      S_Coil( #CONTROL.bENABLE_RFG )
   END_RUNG
   RUNG wire#w1
      S_Coil( #CONTROL.bSETPOINT_ENABLE )
   END_RUNG
   RUNG wire#w1
      R_Coil( #CONTROL.bCW_ACTIVATION )
   END_RUNG
   RUNG wire#w1
      R_Coil( #CONTROL.bCCW_ACTIVATION )
   END_RUNG
   RUNG wire#w1
      S_Coil( #CONTROL.bSP_VALID )
   END_RUNG
   RUNG wire#w1
      S_Coil( #CONTROL.bSP_INVERTED )
   END_RUNG
   RUNG wire#w1
      R_Coil( #CONTROL.bSPARE01 )
   END_RUNG
   RUNG wire#w1
      R_Coil( #CONTROL.bMOTOR_POT_UP )
   END_RUNG
   RUNG wire#w1
      R_Coil( #CONTROL.bMOTOR_POT_DN )
   END_RUNG
   RUNG wire#w1
      R_Coil( #CONTROL.bLOCAL_ACTIVE )
   END_RUNG
   // the same network as SCL:
   IF #STATUS.bMASTER_CONTROL AND NOT #bMajorFault AND #HMI_VFD_Control.bReverseOn AND NOT #HMI_VFD_Control.bForwardOn THEN
       #CONTROL.bON := TRUE;
       #CONTROL.bOFF2 := TRUE;
       #CONTROL.bOFF3 := TRUE;
       #CONTROL.bENABLE_OPERATION := TRUE;
       #CONTROL.bDISABLE_RFG := TRUE;
       #CONTROL.bENABLE_RFG := TRUE;
       #CONTROL.bSETPOINT_ENABLE := TRUE;
       #CONTROL.bCW_ACTIVATION := FALSE;
       #CONTROL.bCCW_ACTIVATION := FALSE;
       #CONTROL.bSP_VALID := TRUE;
       #CONTROL.bSP_INVERTED := TRUE;
       #CONTROL.bSPARE01 := FALSE;
       #CONTROL.bMOTOR_POT_UP := FALSE;
       #CONTROL.bMOTOR_POT_DN := FALSE;
       #CONTROL.bLOCAL_ACTIVE := FALSE;
   END_IF;
END_REGION

REGION Network 49: Set command bits when nothing is commanded, but no faults
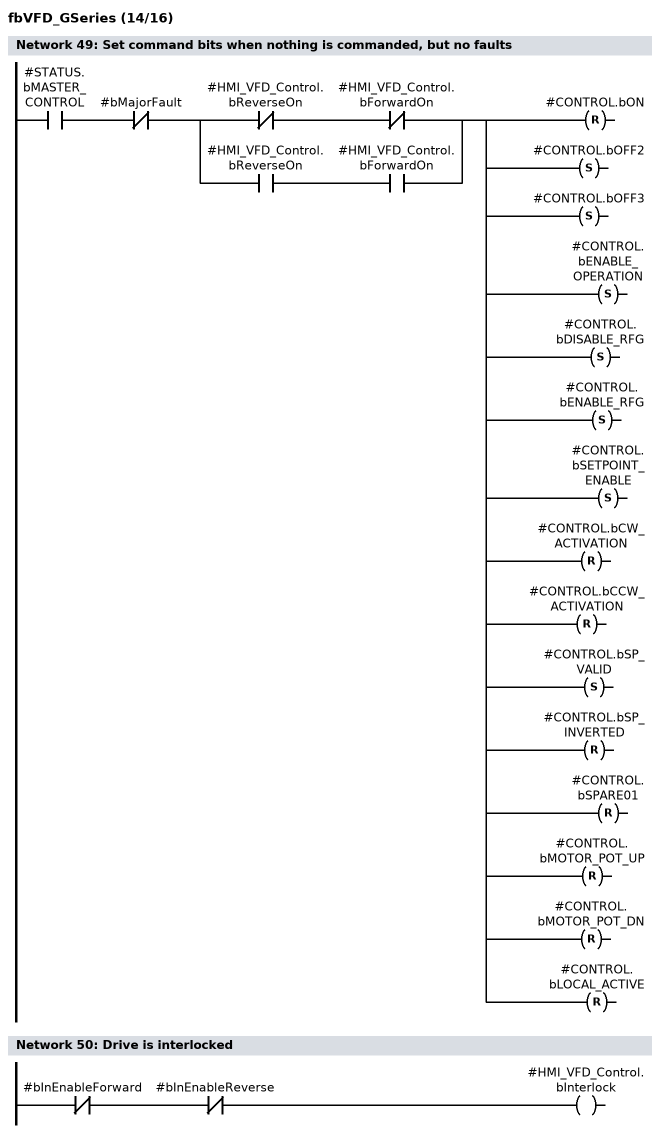
   RUNG wire#powerrail
      Contact( #STATUS.bMASTER_CONTROL )
      I_Contact( #bMajorFault )
      wire#w1
      I_Contact( #HMI_VFD_Control.bReverseOn )
      I_Contact( #HMI_VFD_Control.bForwardOn )
      wire#w2
      R_Coil( #CONTROL.bON )
   END_RUNG
   RUNG wire#w1
      Contact( #HMI_VFD_Control.bReverseOn )
      Contact( #HMI_VFD_Control.bForwardOn )
   END_RUNG wire#w2
   RUNG wire#w2
      S_Coil( #CONTROL.bOFF2 )
   END_RUNG
   RUNG wire#w2
      S_Coil( #CONTROL.bOFF3 )
   END_RUNG
   RUNG wire#w2
      S_Coil( #CONTROL.bENABLE_OPERATION )
   END_RUNG
   RUNG wire#w2
      S_Coil( #CONTROL.bDISABLE_RFG )
   END_RUNG
   RUNG wire#w2
      S_Coil( #CONTROL.bENABLE_RFG )
   END_RUNG
   RUNG wire#w2
      S_Coil( #CONTROL.bSETPOINT_ENABLE )
   END_RUNG
   RUNG wire#w2
      R_Coil( #CONTROL.bCW_ACTIVATION )
   END_RUNG
   RUNG wire#w2
      R_Coil( #CONTROL.bCCW_ACTIVATION )
   END_RUNG
   RUNG wire#w2
      S_Coil( #CONTROL.bSP_VALID )
   END_RUNG
   RUNG wire#w2
      R_Coil( #CONTROL.bSP_INVERTED )
   END_RUNG
   RUNG wire#w2
      R_Coil( #CONTROL.bSPARE01 )
   END_RUNG
   RUNG wire#w2
      R_Coil( #CONTROL.bMOTOR_POT_UP )
   END_RUNG
   RUNG wire#w2
      R_Coil( #CONTROL.bMOTOR_POT_DN )
   END_RUNG
   RUNG wire#w2
      R_Coil( #CONTROL.bLOCAL_ACTIVE )
   END_RUNG
   // the same network as SCL:
   IF #STATUS.bMASTER_CONTROL AND NOT #bMajorFault AND ((NOT #HMI_VFD_Control.bReverseOn AND NOT #HMI_VFD_Control.bForwardOn) OR (#HMI_VFD_Control.bReverseOn AND #HMI_VFD_Control.bForwardOn)) THEN
       #CONTROL.bON := FALSE;
       #CONTROL.bOFF2 := TRUE;
       #CONTROL.bOFF3 := TRUE;
       #CONTROL.bENABLE_OPERATION := TRUE;
       #CONTROL.bDISABLE_RFG := TRUE;
       #CONTROL.bENABLE_RFG := TRUE;
       #CONTROL.bSETPOINT_ENABLE := TRUE;
       #CONTROL.bCW_ACTIVATION := FALSE;
       #CONTROL.bCCW_ACTIVATION := FALSE;
       #CONTROL.bSP_VALID := TRUE;
       #CONTROL.bSP_INVERTED := FALSE;
       #CONTROL.bSPARE01 := FALSE;
       #CONTROL.bMOTOR_POT_UP := FALSE;
       #CONTROL.bMOTOR_POT_DN := FALSE;
       #CONTROL.bLOCAL_ACTIVE := FALSE;
   END_IF;
END_REGION

REGION Network 50: Drive is interlocked
   RUNG wire#powerrail
      I_Contact( #bInEnableForward )
      I_Contact( #bInEnableReverse )
      Coil( #HMI_VFD_Control.bInterlock )
   END_RUNG
   // the same network as SCL:
   #HMI_VFD_Control.bInterlock := NOT #bInEnableForward AND NOT #bInEnableReverse;
END_REGION

REGION Network 51: Set HMI status
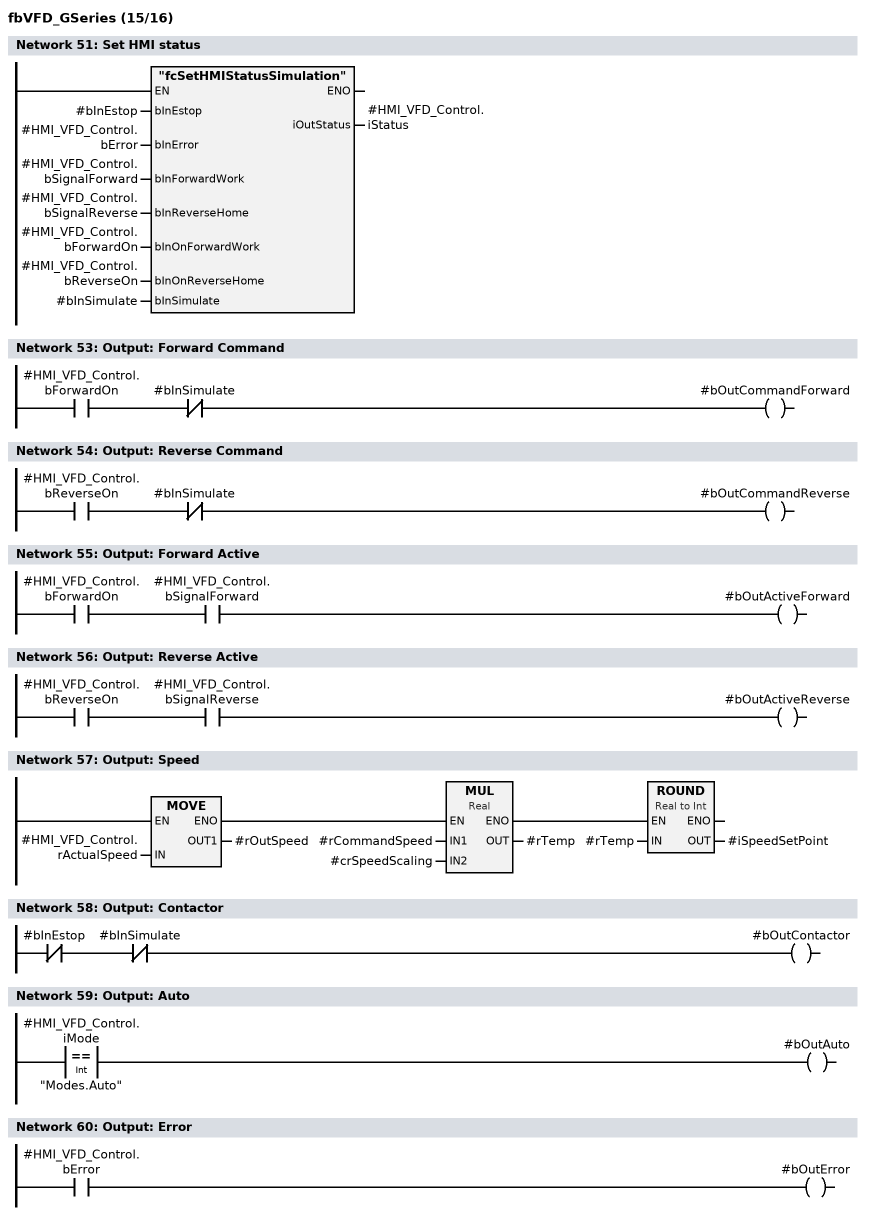
   RUNG wire#powerrail
      "fcSetHMIStatusSimulation"(bInEstop := #bInEstop, bInError := #HMI_VFD_Control.bError, bInForwardWork := #HMI_VFD_Control.bSignalForward, bInReverseHome := #HMI_VFD_Control.bSignalReverse, bInOnForwardWork := #HMI_VFD_Control.bForwardOn, bInOnReverseHome := #HMI_VFD_Control.bReverseOn, bInSimulate := #bInSimulate, iOutStatus => #HMI_VFD_Control.iStatus)
   END_RUNG
   // the same network as SCL:
   "fcSetHMIStatusSimulation"(bInEstop := #bInEstop,
                           bInError := #HMI_VFD_Control.bError,
                           bInForwardWork := #HMI_VFD_Control.bSignalForward,
                           bInReverseHome := #HMI_VFD_Control.bSignalReverse,
                           bInOnForwardWork := #HMI_VFD_Control.bForwardOn,
                           bInOnReverseHome := #HMI_VFD_Control.bReverseOn,
                           bInSimulate := #bInSimulate,
                           iOutStatus => #HMI_VFD_Control.iStatus);
END_REGION

REGION Network 52: --------------------------------------------------------- Outputs ------------------------------------------------------------------
END_REGION

REGION Network 53: Output: Forward Command
   RUNG wire#powerrail
      Contact( #HMI_VFD_Control.bForwardOn )
      I_Contact( #bInSimulate )
      Coil( #bOutCommandForward )
   END_RUNG
   // the same network as SCL:
   #bOutCommandForward := #HMI_VFD_Control.bForwardOn AND NOT #bInSimulate;
END_REGION

REGION Network 54: Output: Reverse Command
   RUNG wire#powerrail
      Contact( #HMI_VFD_Control.bReverseOn )
      I_Contact( #bInSimulate )
      Coil( #bOutCommandReverse )
   END_RUNG
   // the same network as SCL:
   #bOutCommandReverse := #HMI_VFD_Control.bReverseOn AND NOT #bInSimulate;
END_REGION

REGION Network 55: Output: Forward Active
   RUNG wire#powerrail
      Contact( #HMI_VFD_Control.bForwardOn )
      Contact( #HMI_VFD_Control.bSignalForward )
      Coil( #bOutActiveForward )
   END_RUNG
   // the same network as SCL:
   #bOutActiveForward := #HMI_VFD_Control.bForwardOn AND #HMI_VFD_Control.bSignalForward;
END_REGION

REGION Network 56: Output: Reverse Active
   RUNG wire#powerrail
      Contact( #HMI_VFD_Control.bReverseOn )
      Contact( #HMI_VFD_Control.bSignalReverse )
      Coil( #bOutActiveReverse )
   END_RUNG
   // the same network as SCL:
   #bOutActiveReverse := #HMI_VFD_Control.bReverseOn AND #HMI_VFD_Control.bSignalReverse;
END_REGION

REGION Network 57: Output: Speed
   RUNG wire#powerrail
      Move(in := #HMI_VFD_Control.rActualSpeed, out1 => #rOutSpeed)
      { S7_Templates := "SrcType := Real" } Mul(in1 := #rCommandSpeed, in2 := #crSpeedScaling, out => #rTemp)
      { S7_Templates := "[SrcType := Real, DestType := Int]" } Round(in := #rTemp, out => #iSpeedSetPoint)
   END_RUNG
   // the same network as SCL:
   #rOutSpeed := #HMI_VFD_Control.rActualSpeed;
   #rTemp := #rCommandSpeed * #crSpeedScaling;
   #iSpeedSetPoint := ROUND(#rTemp);
END_REGION

REGION Network 58: Output: Contactor
   RUNG wire#powerrail
      I_Contact( #bInEstop )
      I_Contact( #bInSimulate )
      Coil( #bOutContactor )
   END_RUNG
   // the same network as SCL:
   #bOutContactor := NOT #bInEstop AND NOT #bInSimulate;
END_REGION

REGION Network 59: Output: Auto
   RUNG wire#powerrail
      { S7_Templates := "SrcType := Int" } EQ_Contact(in1 := #HMI_VFD_Control.iMode, in2 := "Modes.Auto")
      Coil( #bOutAuto )
   END_RUNG
   // the same network as SCL:
   #bOutAuto := #HMI_VFD_Control.iMode = "Modes.Auto";
END_REGION

REGION Network 60: Output: Error
   RUNG wire#powerrail
      Contact( #HMI_VFD_Control.bError )
      Coil( #bOutError )
   END_RUNG
   // the same network as SCL:
   #bOutError := #HMI_VFD_Control.bError;
END_REGION

REGION Network 61: Output: Control Word
   // assemble control bits into control word
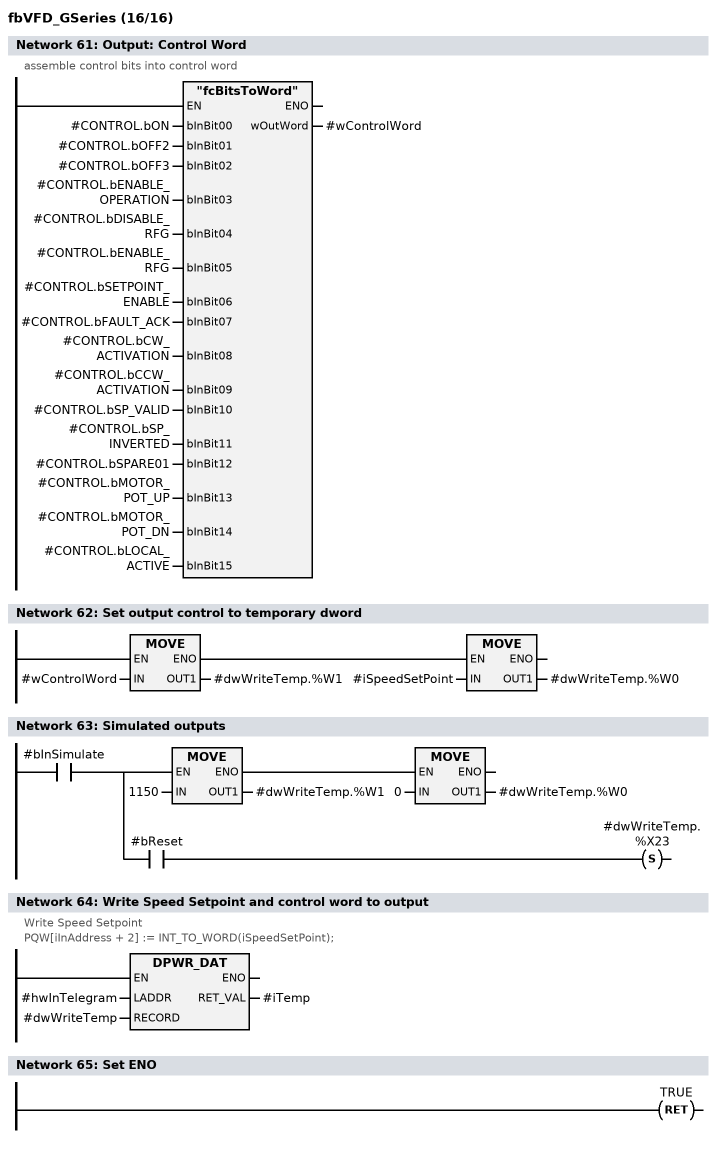
   RUNG wire#powerrail
      "fcBitsToWord"(bInBit00 := #CONTROL.bON, bInBit01 := #CONTROL.bOFF2, bInBit02 := #CONTROL.bOFF3, bInBit03 := #CONTROL.bENABLE_OPERATION, bInBit04 := #CONTROL.bDISABLE_RFG, bInBit05 := #CONTROL.bENABLE_RFG, bInBit06 := #CONTROL.bSETPOINT_ENABLE, bInBit07 := #CONTROL.bFAULT_ACK, bInBit08 := #CONTROL.bCW_ACTIVATION, bInBit09 := #CONTROL.bCCW_ACTIVATION, bInBit10 := #CONTROL.bSP_VALID, bInBit11 := #CONTROL.bSP_INVERTED, bInBit12 := #CONTROL.bSPARE01, bInBit13 := #CONTROL.bMOTOR_POT_UP, bInBit14 := #CONTROL.bMOTOR_POT_DN, bInBit15 := #CONTROL.bLOCAL_ACTIVE, wOutWord => #wControlWord)
   END_RUNG
   // the same network as SCL:
   "fcBitsToWord"(bInBit00 := #CONTROL.bON,
                  bInBit01 := #CONTROL.bOFF2,
                  bInBit02 := #CONTROL.bOFF3,
                  bInBit03 := #CONTROL.bENABLE_OPERATION,
                  bInBit04 := #CONTROL.bDISABLE_RFG,
                  bInBit05 := #CONTROL.bENABLE_RFG,
                  bInBit06 := #CONTROL.bSETPOINT_ENABLE,
                  bInBit07 := #CONTROL.bFAULT_ACK,
                  bInBit08 := #CONTROL.bCW_ACTIVATION,
                  bInBit09 := #CONTROL.bCCW_ACTIVATION,
                  bInBit10 := #CONTROL.bSP_VALID,
                  bInBit11 := #CONTROL.bSP_INVERTED,
                  bInBit12 := #CONTROL.bSPARE01,
                  bInBit13 := #CONTROL.bMOTOR_POT_UP,
                  bInBit14 := #CONTROL.bMOTOR_POT_DN,
                  bInBit15 := #CONTROL.bLOCAL_ACTIVE,
                  wOutWord => #wControlWord);
END_REGION

REGION Network 62: Set output control to temporary dword
   RUNG wire#powerrail
      Move(in := #wControlWord, out1 => #dwWriteTemp.%W1)
      Move(in := #iSpeedSetPoint, out1 => #dwWriteTemp.%W0)
   END_RUNG
   // the same network as SCL:
   #dwWriteTemp.%W1 := #wControlWord;
   #dwWriteTemp.%W0 := #iSpeedSetPoint;
END_REGION

REGION Network 63: Simulated outputs
   RUNG wire#powerrail
      Contact( #bInSimulate )
      wire#w1
      Move(in := 1150, out1 => #dwWriteTemp.%W1)
      Move(in := 0, out1 => #dwWriteTemp.%W0)
   END_RUNG
   RUNG wire#w1
      Contact( #bReset )
      S_Coil( #dwWriteTemp.%X23 )
   END_RUNG
   // the same network as SCL:
   IF #bInSimulate THEN
       #dwWriteTemp.%W1 := 1150;
       #dwWriteTemp.%W0 := 0;
   END_IF;
   IF #bInSimulate AND #bReset THEN #dwWriteTemp.%X23 := TRUE; END_IF;
END_REGION

REGION Network 64: Write Speed Setpoint and control word to output
   // Write Speed Setpoint
   // PQW[iInAddress + 2] := INT_TO_WORD(iSpeedSetPoint);
   #iTemp := DPWR_DAT(LADDR := #hwInTelegram, RECORD := #dwWriteTemp);
END_REGION

REGION Network 65: Set ENO
   RUNG wire#powerrail
      ReturnCoil( TRUE )
   END_RUNG
   // the same network as SCL:
   ENO := TRUE;
   RETURN;
END_REGION
END_FUNCTION_BLOCK

// folder: Resources/fbVFD/Resources/Conversion

FUNCTION "fcBitsToWord" : Void   // FC301, LAD
TITLE = Pack Bits into word
{ S7_Optimized_Access := 'TRUE' }
AUTHOR : DMC
FAMILY : LowLevel
VERSION : 0.1
   VAR_INPUT
      bInBit00 : Bool;   // Bit 0
      bInBit01 : Bool;   // Bit 1
      bInBit02 : Bool;   // Bit 2
      bInBit03 : Bool;   // Bit 3
      bInBit04 : Bool;   // Bit 4
      bInBit05 : Bool;   // Bit 5
      bInBit06 : Bool;   // Bit 6
      bInBit07 : Bool;   // Bit 7
      bInBit08 : Bool;   // Bit 8
      bInBit09 : Bool;   // Bit 9
      bInBit10 : Bool;   // Bit 10
      bInBit11 : Bool;   // Bit 11
      bInBit12 : Bool;   // Bit 12
      bInBit13 : Bool;   // Bit 13
      bInBit14 : Bool;   // Bit 14
      bInBit15 : Bool;   // Bit 15
   END_VAR
   VAR_OUTPUT
      wOutWord : Word;   // Packed Word
   END_VAR
BEGIN

REGION Network 1: Bit0
